   STATUS[908].EXT.ModeBit1 := FALSE;
   STATUS[908].EXT.ModeBit2 := FALSE;
   STATUS[908].EXT.ModeBit3 := FALSE;
   STATUS[908].EXT.BIT19 := FALSE;
   STATUS[908].EXT.BIT20 := FALSE;
   STATUS[908].EXT.AlarmSuppressed := FALSE;
   STATUS[908].EXT.AlarmPrsent := FALSE;
   STATUS[908].EXT.AlarmFailUnAck := FALSE;
   STATUS[908].Status := 0;
   STATUS[908].TimeStamp := 16#0000;
   STATUS[909].VALUE := 0.0;
   STATUS[909].TRIGVALUE := 0.0;
   STATUS[909].EXT.AlarmWarnUnAck := FALSE;
   STATUS[909].EXT.AckRequired := FALSE;
   STATUS[909].EXT.Maintanence := FALSE;
   STATUS[909].EXT.Operation := FALSE;
   STATUS[909].EXT.Forced := FALSE;
   STATUS[909].EXT.BIT29 := FALSE;
   STATUS[909].EXT.BIT30 := FALSE;
   STATUS[909].EXT.BIT31 := FALSE;
   STATUS[909].EXT.ModeBit1 := FALSE;
   STATUS[909].EXT.ModeBit2 := FALSE;
   STATUS[909].EXT.ModeBit3 := FALSE;
   STATUS[909].EXT.BIT19 := FALSE;
   STATUS[909].EXT.BIT20 := FALSE;
   STATUS[909].EXT.AlarmSuppressed := FALSE;
   STATUS[909].EXT.AlarmPrsent := FALSE;
   STATUS[909].EXT.AlarmFailUnAck := FALSE;
   STATUS[909].Status := 0;
   STATUS[909].TimeStamp := 16#0000;
   STATUS[910].VALUE := 0.0;
   STATUS[910].TRIGVALUE := 0.0;
   STATUS[910].EXT.AlarmWarnUnAck := FALSE;
   STATUS[910].EXT.AckRequired := FALSE;
   STATUS[910].EXT.Maintanence := FALSE;
   STATUS[910].EXT.Operation := FALSE;
   STATUS[910].EXT.Forced := FALSE;
   STATUS[910].EXT.BIT29 := FALSE;
   STATUS[910].EXT.BIT30 := FALSE;
   STATUS[910].EXT.BIT31 := FALSE;
   STATUS[910].EXT.ModeBit1 := FALSE;
   STATUS[910].EXT.ModeBit2 := FALSE;
   STATUS[910].EXT.ModeBit3 := FALSE;
   STATUS[910].EXT.BIT19 := FALSE;
   STATUS[910].EXT.BIT20 := FALSE;
   STATUS[910].EXT.AlarmSuppressed := FALSE;
   STATUS[910].EXT.AlarmPrsent := FALSE;
   STATUS[910].EXT.AlarmFailUnAck := FALSE;
   STATUS[910].Status := 0;
   STATUS[910].TimeStamp := 16#0000;
   STATUS[911].VALUE := 0.0;
   STATUS[911].TRIGVALUE := 0.0;
   STATUS[911].EXT.AlarmWarnUnAck := FALSE;
   STATUS[911].EXT.AckRequired := FALSE;
   STATUS[911].EXT.Maintanence := FALSE;
   STATUS[911].EXT.Operation := FALSE;
   STATUS[911].EXT.Forced := FALSE;
   STATUS[911].EXT.BIT29 := FALSE;
   STATUS[911].EXT.BIT30 := FALSE;
   STATUS[911].EXT.BIT31 := FALSE;
   STATUS[911].EXT.ModeBit1 := FALSE;
   STATUS[911].EXT.ModeBit2 := FALSE;
   STATUS[911].EXT.ModeBit3 := FALSE;
   STATUS[911].EXT.BIT19 := FALSE;
   STATUS[911].EXT.BIT20 := FALSE;
   STATUS[911].EXT.AlarmSuppressed := FALSE;
   STATUS[911].EXT.AlarmPrsent := FALSE;
   STATUS[911].EXT.AlarmFailUnAck := FALSE;
   STATUS[911].Status := 0;
   STATUS[911].TimeStamp := 16#0000;
   STATUS[912].VALUE := 0.0;
   STATUS[912].TRIGVALUE := 0.0;
   STATUS[912].EXT.AlarmWarnUnAck := FALSE;
   STATUS[912].EXT.AckRequired := FALSE;
   STATUS[912].EXT.Maintanence := FALSE;
   STATUS[912].EXT.Operation := FALSE;
   STATUS[912].EXT.Forced := FALSE;
   STATUS[912].EXT.BIT29 := FALSE;
   STATUS[912].EXT.BIT30 := FALSE;
   STATUS[912].EXT.BIT31 := FALSE;
   STATUS[912].EXT.ModeBit1 := FALSE;
   STATUS[912].EXT.ModeBit2 := FALSE;
   STATUS[912].EXT.ModeBit3 := FALSE;
   STATUS[912].EXT.BIT19 := FALSE;
   STATUS[912].EXT.BIT20 := FALSE;
   STATUS[912].EXT.AlarmSuppressed := FALSE;
   STATUS[912].EXT.AlarmPrsent := FALSE;
   STATUS[912].EXT.AlarmFailUnAck := FALSE;
   STATUS[912].Status := 0;
   STATUS[912].TimeStamp := 16#0000;
   STATUS[913].VALUE := 0.0;
   STATUS[913].TRIGVALUE := 0.0;
   STATUS[913].EXT.AlarmWarnUnAck := FALSE;
   STATUS[913].EXT.AckRequired := FALSE;
   STATUS[913].EXT.Maintanence := FALSE;
   STATUS[913].EXT.Operation := FALSE;
   STATUS[913].EXT.Forced := FALSE;
   STATUS[913].EXT.BIT29 := FALSE;
   STATUS[913].EXT.BIT30 := FALSE;
   STATUS[913].EXT.BIT31 := FALSE;
   STATUS[913].EXT.ModeBit1 := FALSE;
   STATUS[913].EXT.ModeBit2 := FALSE;
   STATUS[913].EXT.ModeBit3 := FALSE;
   STATUS[913].EXT.BIT19 := FALSE;
   STATUS[913].EXT.BIT20 := FALSE;
   STATUS[913].EXT.AlarmSuppressed := FALSE;
   STATUS[913].EXT.AlarmPrsent := FALSE;
   STATUS[913].EXT.AlarmFailUnAck := FALSE;
   STATUS[913].Status := 0;
   STATUS[913].TimeStamp := 16#0000;
   STATUS[914].VALUE := 0.0;
   STATUS[914].TRIGVALUE := 0.0;
   STATUS[914].EXT.AlarmWarnUnAck := FALSE;
   STATUS[914].EXT.AckRequired := FALSE;
   STATUS[914].EXT.Maintanence := FALSE;
   STATUS[914].EXT.Operation := FALSE;
   STATUS[914].EXT.Forced := FALSE;
   STATUS[914].EXT.BIT29 := FALSE;
   STATUS[914].EXT.BIT30 := FALSE;
   STATUS[914].EXT.BIT31 := FALSE;
   STATUS[914].EXT.ModeBit1 := FALSE;
   STATUS[914].EXT.ModeBit2 := FALSE;
   STATUS[914].EXT.ModeBit3 := FALSE;
   STATUS[914].EXT.BIT19 := FALSE;
   STATUS[914].EXT.BIT20 := FALSE;
   STATUS[914].EXT.AlarmSuppressed := FALSE;
   STATUS[914].EXT.AlarmPrsent := FALSE;
   STATUS[914].EXT.AlarmFailUnAck := FALSE;
   STATUS[914].Status := 0;
   STATUS[914].TimeStamp := 16#0000;
   STATUS[915].VALUE := 0.0;
   STATUS[915].TRIGVALUE := 0.0;
   STATUS[915].EXT.AlarmWarnUnAck := FALSE;
   STATUS[915].EXT.AckRequired := FALSE;
   STATUS[915].EXT.Maintanence := FALSE;
   STATUS[915].EXT.Operation := FALSE;
   STATUS[915].EXT.Forced := FALSE;
   STATUS[915].EXT.BIT29 := FALSE;
   STATUS[915].EXT.BIT30 := FALSE;
   STATUS[915].EXT.BIT31 := FALSE;
   STATUS[915].EXT.ModeBit1 := FALSE;
   STATUS[915].EXT.ModeBit2 := FALSE;
   STATUS[915].EXT.ModeBit3 := FALSE;
   STATUS[915].EXT.BIT19 := FALSE;
   STATUS[915].EXT.BIT20 := FALSE;
   STATUS[915].EXT.AlarmSuppressed := FALSE;
   STATUS[915].EXT.AlarmPrsent := FALSE;
   STATUS[915].EXT.AlarmFailUnAck := FALSE;
   STATUS[915].Status := 0;
   STATUS[915].TimeStamp := 16#0000;
   STATUS[916].VALUE := 0.0;
   STATUS[916].TRIGVALUE := 0.0;
   STATUS[916].EXT.AlarmWarnUnAck := FALSE;
   STATUS[916].EXT.AckRequired := FALSE;
   STATUS[916].EXT.Maintanence := FALSE;
   STATUS[916].EXT.Operation := FALSE;
   STATUS[916].EXT.Forced := FALSE;
   STATUS[916].EXT.BIT29 := FALSE;
   STATUS[916].EXT.BIT30 := FALSE;
   STATUS[916].EXT.BIT31 := FALSE;
   STATUS[916].EXT.ModeBit1 := FALSE;
   STATUS[916].EXT.ModeBit2 := FALSE;
   STATUS[916].EXT.ModeBit3 := FALSE;
   STATUS[916].EXT.BIT19 := FALSE;
   STATUS[916].EXT.BIT20 := FALSE;
   STATUS[916].EXT.AlarmSuppressed := FALSE;
   STATUS[916].EXT.AlarmPrsent := FALSE;
   STATUS[916].EXT.AlarmFailUnAck := FALSE;
   STATUS[916].Status := 0;
   STATUS[916].TimeStamp := 16#0000;
   STATUS[917].VALUE := 0.0;
   STATUS[917].TRIGVALUE := 0.0;
   STATUS[917].EXT.AlarmWarnUnAck := FALSE;
   STATUS[917].EXT.AckRequired := FALSE;
   STATUS[917].EXT.Maintanence := FALSE;
   STATUS[917].EXT.Operation := FALSE;
   STATUS[917].EXT.Forced := FALSE;
   STATUS[917].EXT.BIT29 := FALSE;
   STATUS[917].EXT.BIT30 := FALSE;
   STATUS[917].EXT.BIT31 := FALSE;
   STATUS[917].EXT.ModeBit1 := FALSE;
   STATUS[917].EXT.ModeBit2 := FALSE;
   STATUS[917].EXT.ModeBit3 := FALSE;
   STATUS[917].EXT.BIT19 := FALSE;
   STATUS[917].EXT.BIT20 := FALSE;
   STATUS[917].EXT.AlarmSuppressed := FALSE;
   STATUS[917].EXT.AlarmPrsent := FALSE;
   STATUS[917].EXT.AlarmFailUnAck := FALSE;
   STATUS[917].Status := 0;
   STATUS[917].TimeStamp := 16#0000;
   STATUS[918].VALUE := 0.0;
   STATUS[918].TRIGVALUE := 0.0;
   STATUS[918].EXT.AlarmWarnUnAck := FALSE;
   STATUS[918].EXT.AckRequired := FALSE;
   STATUS[918].EXT.Maintanence := FALSE;
   STATUS[918].EXT.Operation := FALSE;
   STATUS[918].EXT.Forced := FALSE;
   STATUS[918].EXT.BIT29 := FALSE;
   STATUS[918].EXT.BIT30 := FALSE;
   STATUS[918].EXT.BIT31 := FALSE;
   STATUS[918].EXT.ModeBit1 := FALSE;
   STATUS[918].EXT.ModeBit2 := FALSE;
   STATUS[918].EXT.ModeBit3 := FALSE;
   STATUS[918].EXT.BIT19 := FALSE;
   STATUS[918].EXT.BIT20 := FALSE;
   STATUS[918].EXT.AlarmSuppressed := FALSE;
   STATUS[918].EXT.AlarmPrsent := FALSE;
   STATUS[918].EXT.AlarmFailUnAck := FALSE;
   STATUS[918].Status := 0;
   STATUS[918].TimeStamp := 16#0000;
   STATUS[919].VALUE := 0.0;
   STATUS[919].TRIGVALUE := 0.0;
   STATUS[919].EXT.AlarmWarnUnAck := FALSE;
   STATUS[919].EXT.AckRequired := FALSE;
   STATUS[919].EXT.Maintanence := FALSE;
   STATUS[919].EXT.Operation := FALSE;
   STATUS[919].EXT.Forced := FALSE;
   STATUS[919].EXT.BIT29 := FALSE;
   STATUS[919].EXT.BIT30 := FALSE;
   STATUS[919].EXT.BIT31 := FALSE;
   STATUS[919].EXT.ModeBit1 := FALSE;
   STATUS[919].EXT.ModeBit2 := FALSE;
   STATUS[919].EXT.ModeBit3 := FALSE;
   STATUS[919].EXT.BIT19 := FALSE;
   STATUS[919].EXT.BIT20 := FALSE;
   STATUS[919].EXT.AlarmSuppressed := FALSE;
   STATUS[919].EXT.AlarmPrsent := FALSE;
   STATUS[919].EXT.AlarmFailUnAck := FALSE;
   STATUS[919].Status := 0;
   STATUS[919].TimeStamp := 16#0000;
   STATUS[920].VALUE := 0.0;
   STATUS[920].TRIGVALUE := 0.0;
   STATUS[920].EXT.AlarmWarnUnAck := FALSE;
   STATUS[920].EXT.AckRequired := FALSE;
   STATUS[920].EXT.Maintanence := FALSE;
   STATUS[920].EXT.Operation := FALSE;
   STATUS[920].EXT.Forced := FALSE;
   STATUS[920].EXT.BIT29 := FALSE;
   STATUS[920].EXT.BIT30 := FALSE;
   STATUS[920].EXT.BIT31 := FALSE;
   STATUS[920].EXT.ModeBit1 := FALSE;
   STATUS[920].EXT.ModeBit2 := FALSE;
   STATUS[920].EXT.ModeBit3 := FALSE;
   STATUS[920].EXT.BIT19 := FALSE;
   STATUS[920].EXT.BIT20 := FALSE;
   STATUS[920].EXT.AlarmSuppressed := FALSE;
   STATUS[920].EXT.AlarmPrsent := FALSE;
   STATUS[920].EXT.AlarmFailUnAck := FALSE;
   STATUS[920].Status := 0;
   STATUS[920].TimeStamp := 16#0000;
   STATUS[921].VALUE := 0.0;
   STATUS[921].TRIGVALUE := 0.0;
   STATUS[921].EXT.AlarmWarnUnAck := FALSE;
   STATUS[921].EXT.AckRequired := FALSE;
   STATUS[921].EXT.Maintanence := FALSE;
   STATUS[921].EXT.Operation := FALSE;
   STATUS[921].EXT.Forced := FALSE;
   STATUS[921].EXT.BIT29 := FALSE;
   STATUS[921].EXT.BIT30 := FALSE;
   STATUS[921].EXT.BIT31 := FALSE;
   STATUS[921].EXT.ModeBit1 := FALSE;
   STATUS[921].EXT.ModeBit2 := FALSE;
   STATUS[921].EXT.ModeBit3 := FALSE;
   STATUS[921].EXT.BIT19 := FALSE;
   STATUS[921].EXT.BIT20 := FALSE;
   STATUS[921].EXT.AlarmSuppressed := FALSE;
   STATUS[921].EXT.AlarmPrsent := FALSE;
   STATUS[921].EXT.AlarmFailUnAck := FALSE;
   STATUS[921].Status := 0;
   STATUS[921].TimeStamp := 16#0000;
   STATUS[922].VALUE := 0.0;
   STATUS[922].TRIGVALUE := 0.0;
   STATUS[922].EXT.AlarmWarnUnAck := FALSE;
   STATUS[922].EXT.AckRequired := FALSE;
   STATUS[922].EXT.Maintanence := FALSE;
   STATUS[922].EXT.Operation := FALSE;
   STATUS[922].EXT.Forced := FALSE;
   STATUS[922].EXT.BIT29 := FALSE;
   STATUS[922].EXT.BIT30 := FALSE;
   STATUS[922].EXT.BIT31 := FALSE;
   STATUS[922].EXT.ModeBit1 := FALSE;
   STATUS[922].EXT.ModeBit2 := FALSE;
   STATUS[922].EXT.ModeBit3 := FALSE;
   STATUS[922].EXT.BIT19 := FALSE;
   STATUS[922].EXT.BIT20 := FALSE;
   STATUS[922].EXT.AlarmSuppressed := FALSE;
   STATUS[922].EXT.AlarmPrsent := FALSE;
   STATUS[922].EXT.AlarmFailUnAck := FALSE;
   STATUS[922].Status := 0;
   STATUS[922].TimeStamp := 16#0000;
   STATUS[923].VALUE := 0.0;
   STATUS[923].TRIGVALUE := 0.0;
   STATUS[923].EXT.AlarmWarnUnAck := FALSE;
   STATUS[923].EXT.AckRequired := FALSE;
   STATUS[923].EXT.Maintanence := FALSE;
   STATUS[923].EXT.Operation := FALSE;
   STATUS[923].EXT.Forced := FALSE;
   STATUS[923].EXT.BIT29 := FALSE;
   STATUS[923].EXT.BIT30 := FALSE;
   STATUS[923].EXT.BIT31 := FALSE;
   STATUS[923].EXT.ModeBit1 := FALSE;
   STATUS[923].EXT.ModeBit2 := FALSE;
   STATUS[923].EXT.ModeBit3 := FALSE;
   STATUS[923].EXT.BIT19 := FALSE;
   STATUS[923].EXT.BIT20 := FALSE;
   STATUS[923].EXT.AlarmSuppressed := FALSE;
   STATUS[923].EXT.AlarmPrsent := FALSE;
   STATUS[923].EXT.AlarmFailUnAck := FALSE;
   STATUS[923].Status := 0;
   STATUS[923].TimeStamp := 16#0000;
   STATUS[924].VALUE := 0.0;
   STATUS[924].TRIGVALUE := 0.0;
   STATUS[924].EXT.AlarmWarnUnAck := FALSE;
   STATUS[924].EXT.AckRequired := FALSE;
   STATUS[924].EXT.Maintanence := FALSE;
   STATUS[924].EXT.Operation := FALSE;
   STATUS[924].EXT.Forced := FALSE;
   STATUS[924].EXT.BIT29 := FALSE;
   STATUS[924].EXT.BIT30 := FALSE;
   STATUS[924].EXT.BIT31 := FALSE;
   STATUS[924].EXT.ModeBit1 := FALSE;
   STATUS[924].EXT.ModeBit2 := FALSE;
   STATUS[924].EXT.ModeBit3 := FALSE;
   STATUS[924].EXT.BIT19 := FALSE;
   STATUS[924].EXT.BIT20 := FALSE;
   STATUS[924].EXT.AlarmSuppressed := FALSE;
   STATUS[924].EXT.AlarmPrsent := FALSE;
   STATUS[924].EXT.AlarmFailUnAck := FALSE;
   STATUS[924].Status := 0;
   STATUS[924].TimeStamp := 16#0000;
   STATUS[925].VALUE := 0.0;
   STATUS[925].TRIGVALUE := 0.0;
   STATUS[925].EXT.AlarmWarnUnAck := FALSE;
   STATUS[925].EXT.AckRequired := FALSE;
   STATUS[925].EXT.Maintanence := FALSE;
   STATUS[925].EXT.Operation := FALSE;
   STATUS[925].EXT.Forced := FALSE;
   STATUS[925].EXT.BIT29 := FALSE;
   STATUS[925].EXT.BIT30 := FALSE;
   STATUS[925].EXT.BIT31 := FALSE;
   STATUS[925].EXT.ModeBit1 := FALSE;
   STATUS[925].EXT.ModeBit2 := FALSE;
   STATUS[925].EXT.ModeBit3 := FALSE;
   STATUS[925].EXT.BIT19 := FALSE;
   STATUS[925].EXT.BIT20 := FALSE;
   STATUS[925].EXT.AlarmSuppressed := FALSE;
   STATUS[925].EXT.AlarmPrsent := FALSE;
   STATUS[925].EXT.AlarmFailUnAck := FALSE;
   STATUS[925].Status := 0;
   STATUS[925].TimeStamp := 16#0000;
   STATUS[926].VALUE := 0.0;
   STATUS[926].TRIGVALUE := 0.0;
   STATUS[926].EXT.AlarmWarnUnAck := FALSE;
   STATUS[926].EXT.AckRequired := FALSE;
   STATUS[926].EXT.Maintanence := FALSE;
   STATUS[926].EXT.Operation := FALSE;
   STATUS[926].EXT.Forced := FALSE;
   STATUS[926].EXT.BIT29 := FALSE;
   STATUS[926].EXT.BIT30 := FALSE;
   STATUS[926].EXT.BIT31 := FALSE;
   STATUS[926].EXT.ModeBit1 := FALSE;
   STATUS[926].EXT.ModeBit2 := FALSE;
   STATUS[926].EXT.ModeBit3 := FALSE;
   STATUS[926].EXT.BIT19 := FALSE;
   STATUS[926].EXT.BIT20 := FALSE;
   STATUS[926].EXT.AlarmSuppressed := FALSE;
   STATUS[926].EXT.AlarmPrsent := FALSE;
   STATUS[926].EXT.AlarmFailUnAck := FALSE;
   STATUS[926].Status := 0;
   STATUS[926].TimeStamp := 16#0000;
   STATUS[927].VALUE := 0.0;
   STATUS[927].TRIGVALUE := 0.0;
   STATUS[927].EXT.AlarmWarnUnAck := FALSE;
   STATUS[927].EXT.AckRequired := FALSE;
   STATUS[927].EXT.Maintanence := FALSE;
   STATUS[927].EXT.Operation := FALSE;
   STATUS[927].EXT.Forced := FALSE;
   STATUS[927].EXT.BIT29 := FALSE;
   STATUS[927].EXT.BIT30 := FALSE;
   STATUS[927].EXT.BIT31 := FALSE;
   STATUS[927].EXT.ModeBit1 := FALSE;
   STATUS[927].EXT.ModeBit2 := FALSE;
   STATUS[927].EXT.ModeBit3 := FALSE;
   STATUS[927].EXT.BIT19 := FALSE;
   STATUS[927].EXT.BIT20 := FALSE;
   STATUS[927].EXT.AlarmSuppressed := FALSE;
   STATUS[927].EXT.AlarmPrsent := FALSE;
   STATUS[927].EXT.AlarmFailUnAck := FALSE;
   STATUS[927].Status := 0;
   STATUS[927].TimeStamp := 16#0000;
   STATUS[928].VALUE := 0.0;
   STATUS[928].TRIGVALUE := 0.0;
   STATUS[928].EXT.AlarmWarnUnAck := FALSE;
   STATUS[928].EXT.AckRequired := FALSE;
   STATUS[928].EXT.Maintanence := FALSE;
   STATUS[928].EXT.Operation := FALSE;
   STATUS[928].EXT.Forced := FALSE;
   STATUS[928].EXT.BIT29 := FALSE;
   STATUS[928].EXT.BIT30 := FALSE;
   STATUS[928].EXT.BIT31 := FALSE;
   STATUS[928].EXT.ModeBit1 := FALSE;
   STATUS[928].EXT.ModeBit2 := FALSE;
   STATUS[928].EXT.ModeBit3 := FALSE;
   STATUS[928].EXT.BIT19 := FALSE;
   STATUS[928].EXT.BIT20 := FALSE;
   STATUS[928].EXT.AlarmSuppressed := FALSE;
   STATUS[928].EXT.AlarmPrsent := FALSE;
   STATUS[928].EXT.AlarmFailUnAck := FALSE;
   STATUS[928].Status := 0;
   STATUS[928].TimeStamp := 16#0000;
   STATUS[929].VALUE := 0.0;
   STATUS[929].TRIGVALUE := 0.0;
   STATUS[929].EXT.AlarmWarnUnAck := FALSE;
   STATUS[929].EXT.AckRequired := FALSE;
   STATUS[929].EXT.Maintanence := FALSE;
   STATUS[929].EXT.Operation := FALSE;
   STATUS[929].EXT.Forced := FALSE;
   STATUS[929].EXT.BIT29 := FALSE;
   STATUS[929].EXT.BIT30 := FALSE;
   STATUS[929].EXT.BIT31 := FALSE;
   STATUS[929].EXT.ModeBit1 := FALSE;
   STATUS[929].EXT.ModeBit2 := FALSE;
   STATUS[929].EXT.ModeBit3 := FALSE;
   STATUS[929].EXT.BIT19 := FALSE;
   STATUS[929].EXT.BIT20 := FALSE;
   STATUS[929].EXT.AlarmSuppressed := FALSE;
   STATUS[929].EXT.AlarmPrsent := FALSE;
   STATUS[929].EXT.AlarmFailUnAck := FALSE;
   STATUS[929].Status := 0;
   STATUS[929].TimeStamp := 16#0000;
   STATUS[930].VALUE := 0.0;
   STATUS[930].TRIGVALUE := 0.0;
   STATUS[930].EXT.AlarmWarnUnAck := FALSE;
   STATUS[930].EXT.AckRequired := FALSE;
   STATUS[930].EXT.Maintanence := FALSE;
   STATUS[930].EXT.Operation := FALSE;
   STATUS[930].EXT.Forced := FALSE;
   STATUS[930].EXT.BIT29 := FALSE;
   STATUS[930].EXT.BIT30 := FALSE;
   STATUS[930].EXT.BIT31 := FALSE;
   STATUS[930].EXT.ModeBit1 := FALSE;
   STATUS[930].EXT.ModeBit2 := FALSE;
   STATUS[930].EXT.ModeBit3 := FALSE;
   STATUS[930].EXT.BIT19 := FALSE;
   STATUS[930].EXT.BIT20 := FALSE;
   STATUS[930].EXT.AlarmSuppressed := FALSE;
   STATUS[930].EXT.AlarmPrsent := FALSE;
   STATUS[930].EXT.AlarmFailUnAck := FALSE;
   STATUS[930].Status := 0;
   STATUS[930].TimeStamp := 16#0000;
   STATUS[931].VALUE := 0.0;
   STATUS[931].TRIGVALUE := 0.0;
   STATUS[931].EXT.AlarmWarnUnAck := FALSE;
   STATUS[931].EXT.AckRequired := FALSE;
   STATUS[931].EXT.Maintanence := FALSE;
   STATUS[931].EXT.Operation := FALSE;
   STATUS[931].EXT.Forced := FALSE;
   STATUS[931].EXT.BIT29 := FALSE;
   STATUS[931].EXT.BIT30 := FALSE;
   STATUS[931].EXT.BIT31 := FALSE;
   STATUS[931].EXT.ModeBit1 := FALSE;
   STATUS[931].EXT.ModeBit2 := FALSE;
   STATUS[931].EXT.ModeBit3 := FALSE;
   STATUS[931].EXT.BIT19 := FALSE;
   STATUS[931].EXT.BIT20 := FALSE;
   STATUS[931].EXT.AlarmSuppressed := FALSE;
   STATUS[931].EXT.AlarmPrsent := FALSE;
   STATUS[931].EXT.AlarmFailUnAck := FALSE;
   STATUS[931].Status := 0;
   STATUS[931].TimeStamp := 16#0000;
   STATUS[932].VALUE := 0.0;
   STATUS[932].TRIGVALUE := 0.0;
   STATUS[932].EXT.AlarmWarnUnAck := FALSE;
   STATUS[932].EXT.AckRequired := FALSE;
   STATUS[932].EXT.Maintanence := FALSE;
   STATUS[932].EXT.Operation := FALSE;
   STATUS[932].EXT.Forced := FALSE;
   STATUS[932].EXT.BIT29 := FALSE;
   STATUS[932].EXT.BIT30 := FALSE;
   STATUS[932].EXT.BIT31 := FALSE;
   STATUS[932].EXT.ModeBit1 := FALSE;
   STATUS[932].EXT.ModeBit2 := FALSE;
   STATUS[932].EXT.ModeBit3 := FALSE;
   STATUS[932].EXT.BIT19 := FALSE;
   STATUS[932].EXT.BIT20 := FALSE;
   STATUS[932].EXT.AlarmSuppressed := FALSE;
   STATUS[932].EXT.AlarmPrsent := FALSE;
   STATUS[932].EXT.AlarmFailUnAck := FALSE;
   STATUS[932].Status := 0;
   STATUS[932].TimeStamp := 16#0000;
   STATUS[933].VALUE := 0.0;
   STATUS[933].TRIGVALUE := 0.0;
   STATUS[933].EXT.AlarmWarnUnAck := FALSE;
   STATUS[933].EXT.AckRequired := FALSE;
   STATUS[933].EXT.Maintanence := FALSE;
   STATUS[933].EXT.Operation := FALSE;
   STATUS[933].EXT.Forced := FALSE;
   STATUS[933].EXT.BIT29 := FALSE;
   STATUS[933].EXT.BIT30 := FALSE;
   STATUS[933].EXT.BIT31 := FALSE;
   STATUS[933].EXT.ModeBit1 := FALSE;
   STATUS[933].EXT.ModeBit2 := FALSE;
   STATUS[933].EXT.ModeBit3 := FALSE;
   STATUS[933].EXT.BIT19 := FALSE;
   STATUS[933].EXT.BIT20 := FALSE;
   STATUS[933].EXT.AlarmSuppressed := FALSE;
   STATUS[933].EXT.AlarmPrsent := FALSE;
   STATUS[933].EXT.AlarmFailUnAck := FALSE;
   STATUS[933].Status := 0;
   STATUS[933].TimeStamp := 16#0000;
   STATUS[934].VALUE := 0.0;
   STATUS[934].TRIGVALUE := 0.0;
   STATUS[934].EXT.AlarmWarnUnAck := FALSE;
   STATUS[934].EXT.AckRequired := FALSE;
   STATUS[934].EXT.Maintanence := FALSE;
   STATUS[934].EXT.Operation := FALSE;
   STATUS[934].EXT.Forced := FALSE;
   STATUS[934].EXT.BIT29 := FALSE;
   STATUS[934].EXT.BIT30 := FALSE;
   STATUS[934].EXT.BIT31 := FALSE;
   STATUS[934].EXT.ModeBit1 := FALSE;
   STATUS[934].EXT.ModeBit2 := FALSE;
   STATUS[934].EXT.ModeBit3 := FALSE;
   STATUS[934].EXT.BIT19 := FALSE;
   STATUS[934].EXT.BIT20 := FALSE;
   STATUS[934].EXT.AlarmSuppressed := FALSE;
   STATUS[934].EXT.AlarmPrsent := FALSE;
   STATUS[934].EXT.AlarmFailUnAck := FALSE;
   STATUS[934].Status := 0;
   STATUS[934].TimeStamp := 16#0000;
   STATUS[935].VALUE := 0.0;
   STATUS[935].TRIGVALUE := 0.0;
   STATUS[935].EXT.AlarmWarnUnAck := FALSE;
   STATUS[935].EXT.AckRequired := FALSE;
   STATUS[935].EXT.Maintanence := FALSE;
   STATUS[935].EXT.Operation := FALSE;
   STATUS[935].EXT.Forced := FALSE;
   STATUS[935].EXT.BIT29 := FALSE;
   STATUS[935].EXT.BIT30 := FALSE;
   STATUS[935].EXT.BIT31 := FALSE;
   STATUS[935].EXT.ModeBit1 := FALSE;
   STATUS[935].EXT.ModeBit2 := FALSE;
   STATUS[935].EXT.ModeBit3 := FALSE;
   STATUS[935].EXT.BIT19 := FALSE;
   STATUS[935].EXT.BIT20 := FALSE;
   STATUS[935].EXT.AlarmSuppressed := FALSE;
   STATUS[935].EXT.AlarmPrsent := FALSE;
   STATUS[935].EXT.AlarmFailUnAck := FALSE;
   STATUS[935].Status := 0;
   STATUS[935].TimeStamp := 16#0000;
   STATUS[936].VALUE := 0.0;
   STATUS[936].TRIGVALUE := 0.0;
   STATUS[936].EXT.AlarmWarnUnAck := FALSE;
   STATUS[936].EXT.AckRequired := FALSE;
   STATUS[936].EXT.Maintanence := FALSE;
   STATUS[936].EXT.Operation := FALSE;
   STATUS[936].EXT.Forced := FALSE;
   STATUS[936].EXT.BIT29 := FALSE;
   STATUS[936].EXT.BIT30 := FALSE;
   STATUS[936].EXT.BIT31 := FALSE;
   STATUS[936].EXT.ModeBit1 := FALSE;
   STATUS[936].EXT.ModeBit2 := FALSE;
   STATUS[936].EXT.ModeBit3 := FALSE;
   STATUS[936].EXT.BIT19 := FALSE;
   STATUS[936].EXT.BIT20 := FALSE;
   STATUS[936].EXT.AlarmSuppressed := FALSE;
   STATUS[936].EXT.AlarmPrsent := FALSE;
   STATUS[936].EXT.AlarmFailUnAck := FALSE;
   STATUS[936].Status := 0;
   STATUS[936].TimeStamp := 16#0000;
   STATUS[937].VALUE := 0.0;
   STATUS[937].TRIGVALUE := 0.0;
   STATUS[937].EXT.AlarmWarnUnAck := FALSE;
   STATUS[937].EXT.AckRequired := FALSE;
   STATUS[937].EXT.Maintanence := FALSE;
   STATUS[937].EXT.Operation := FALSE;
   STATUS[937].EXT.Forced := FALSE;
   STATUS[937].EXT.BIT29 := FALSE;
   STATUS[937].EXT.BIT30 := FALSE;
   STATUS[937].EXT.BIT31 := FALSE;
   STATUS[937].EXT.ModeBit1 := FALSE;
   STATUS[937].EXT.ModeBit2 := FALSE;
   STATUS[937].EXT.ModeBit3 := FALSE;
   STATUS[937].EXT.BIT19 := FALSE;
   STATUS[937].EXT.BIT20 := FALSE;
   STATUS[937].EXT.AlarmSuppressed := FALSE;
   STATUS[937].EXT.AlarmPrsent := FALSE;
   STATUS[937].EXT.AlarmFailUnAck := FALSE;
   STATUS[937].Status := 0;
   STATUS[937].TimeStamp := 16#0000;
   STATUS[938].VALUE := 0.0;
   STATUS[938].TRIGVALUE := 0.0;
   STATUS[938].EXT.AlarmWarnUnAck := FALSE;
   STATUS[938].EXT.AckRequired := FALSE;
   STATUS[938].EXT.Maintanence := FALSE;
   STATUS[938].EXT.Operation := FALSE;
   STATUS[938].EXT.Forced := FALSE;
   STATUS[938].EXT.BIT29 := FALSE;
   STATUS[938].EXT.BIT30 := FALSE;
   STATUS[938].EXT.BIT31 := FALSE;
   STATUS[938].EXT.ModeBit1 := FALSE;
   STATUS[938].EXT.ModeBit2 := FALSE;
   STATUS[938].EXT.ModeBit3 := FALSE;
   STATUS[938].EXT.BIT19 := FALSE;
   STATUS[938].EXT.BIT20 := FALSE;
   STATUS[938].EXT.AlarmSuppressed := FALSE;
   STATUS[938].EXT.AlarmPrsent := FALSE;
   STATUS[938].EXT.AlarmFailUnAck := FALSE;
   STATUS[938].Status := 0;
   STATUS[938].TimeStamp := 16#0000;
   STATUS[939].VALUE := 0.0;
   STATUS[939].TRIGVALUE := 0.0;
   STATUS[939].EXT.AlarmWarnUnAck := FALSE;
   STATUS[939].EXT.AckRequired := FALSE;
   STATUS[939].EXT.Maintanence := FALSE;
   STATUS[939].EXT.Operation := FALSE;
   STATUS[939].EXT.Forced := FALSE;
   STATUS[939].EXT.BIT29 := FALSE;
   STATUS[939].EXT.BIT30 := FALSE;
   STATUS[939].EXT.BIT31 := FALSE;
   STATUS[939].EXT.ModeBit1 := FALSE;
   STATUS[939].EXT.ModeBit2 := FALSE;
   STATUS[939].EXT.ModeBit3 := FALSE;
   STATUS[939].EXT.BIT19 := FALSE;
   STATUS[939].EXT.BIT20 := FALSE;
   STATUS[939].EXT.AlarmSuppressed := FALSE;
   STATUS[939].EXT.AlarmPrsent := FALSE;
   STATUS[939].EXT.AlarmFailUnAck := FALSE;
   STATUS[939].Status := 0;
   STATUS[939].TimeStamp := 16#0000;
   STATUS[940].VALUE := 0.0;
   STATUS[940].TRIGVALUE := 0.0;
   STATUS[940].EXT.AlarmWarnUnAck := FALSE;
   STATUS[940].EXT.AckRequired := FALSE;
   STATUS[940].EXT.Maintanence := FALSE;
   STATUS[940].EXT.Operation := FALSE;
   STATUS[940].EXT.Forced := FALSE;
   STATUS[940].EXT.BIT29 := FALSE;
   STATUS[940].EXT.BIT30 := FALSE;
   STATUS[940].EXT.BIT31 := FALSE;
   STATUS[940].EXT.ModeBit1 := FALSE;
   STATUS[940].EXT.ModeBit2 := FALSE;
   STATUS[940].EXT.ModeBit3 := FALSE;
   STATUS[940].EXT.BIT19 := FALSE;
   STATUS[940].EXT.BIT20 := FALSE;
   STATUS[940].EXT.AlarmSuppressed := FALSE;
   STATUS[940].EXT.AlarmPrsent := FALSE;
   STATUS[940].EXT.AlarmFailUnAck := FALSE;
   STATUS[940].Status := 0;
   STATUS[940].TimeStamp := 16#0000;
   STATUS[941].VALUE := 0.0;
   STATUS[941].TRIGVALUE := 0.0;
   STATUS[941].EXT.AlarmWarnUnAck := FALSE;
   STATUS[941].EXT.AckRequired := FALSE;
   STATUS[941].EXT.Maintanence := FALSE;
   STATUS[941].EXT.Operation := FALSE;
   STATUS[941].EXT.Forced := FALSE;
   STATUS[941].EXT.BIT29 := FALSE;
   STATUS[941].EXT.BIT30 := FALSE;
   STATUS[941].EXT.BIT31 := FALSE;
   STATUS[941].EXT.ModeBit1 := FALSE;
   STATUS[941].EXT.ModeBit2 := FALSE;
   STATUS[941].EXT.ModeBit3 := FALSE;
   STATUS[941].EXT.BIT19 := FALSE;
   STATUS[941].EXT.BIT20 := FALSE;
   STATUS[941].EXT.AlarmSuppressed := FALSE;
   STATUS[941].EXT.AlarmPrsent := FALSE;
   STATUS[941].EXT.AlarmFailUnAck := FALSE;
   STATUS[941].Status := 0;
   STATUS[941].TimeStamp := 16#0000;
   STATUS[942].VALUE := 0.0;
   STATUS[942].TRIGVALUE := 0.0;
   STATUS[942].EXT.AlarmWarnUnAck := FALSE;
   STATUS[942].EXT.AckRequired := FALSE;
   STATUS[942].EXT.Maintanence := FALSE;
   STATUS[942].EXT.Operation := FALSE;
   STATUS[942].EXT.Forced := FALSE;
   STATUS[942].EXT.BIT29 := FALSE;
   STATUS[942].EXT.BIT30 := FALSE;
   STATUS[942].EXT.BIT31 := FALSE;
   STATUS[942].EXT.ModeBit1 := FALSE;
   STATUS[942].EXT.ModeBit2 := FALSE;
   STATUS[942].EXT.ModeBit3 := FALSE;
   STATUS[942].EXT.BIT19 := FALSE;
   STATUS[942].EXT.BIT20 := FALSE;
   STATUS[942].EXT.AlarmSuppressed := FALSE;
   STATUS[942].EXT.AlarmPrsent := FALSE;
   STATUS[942].EXT.AlarmFailUnAck := FALSE;
   STATUS[942].Status := 0;
   STATUS[942].TimeStamp := 16#0000;
   STATUS[943].VALUE := 0.0;
   STATUS[943].TRIGVALUE := 0.0;
   STATUS[943].EXT.AlarmWarnUnAck := FALSE;
   STATUS[943].EXT.AckRequired := FALSE;
   STATUS[943].EXT.Maintanence := FALSE;
   STATUS[943].EXT.Operation := FALSE;
   STATUS[943].EXT.Forced := FALSE;
   STATUS[943].EXT.BIT29 := FALSE;
   STATUS[943].EXT.BIT30 := FALSE;
   STATUS[943].EXT.BIT31 := FALSE;
   STATUS[943].EXT.ModeBit1 := FALSE;
   STATUS[943].EXT.ModeBit2 := FALSE;
   STATUS[943].EXT.ModeBit3 := FALSE;
   STATUS[943].EXT.BIT19 := FALSE;
   STATUS[943].EXT.BIT20 := FALSE;
   STATUS[943].EXT.AlarmSuppressed := FALSE;
   STATUS[943].EXT.AlarmPrsent := FALSE;
   STATUS[943].EXT.AlarmFailUnAck := FALSE;
   STATUS[943].Status := 0;
   STATUS[943].TimeStamp := 16#0000;
   STATUS[944].VALUE := 0.0;
   STATUS[944].TRIGVALUE := 0.0;
   STATUS[944].EXT.AlarmWarnUnAck := FALSE;
   STATUS[944].EXT.AckRequired := FALSE;
   STATUS[944].EXT.Maintanence := FALSE;
   STATUS[944].EXT.Operation := FALSE;
   STATUS[944].EXT.Forced := FALSE;
   STATUS[944].EXT.BIT29 := FALSE;
   STATUS[944].EXT.BIT30 := FALSE;
   STATUS[944].EXT.BIT31 := FALSE;
   STATUS[944].EXT.ModeBit1 := FALSE;
   STATUS[944].EXT.ModeBit2 := FALSE;
   STATUS[944].EXT.ModeBit3 := FALSE;
   STATUS[944].EXT.BIT19 := FALSE;
   STATUS[944].EXT.BIT20 := FALSE;
   STATUS[944].EXT.AlarmSuppressed := FALSE;
   STATUS[944].EXT.AlarmPrsent := FALSE;
   STATUS[944].EXT.AlarmFailUnAck := FALSE;
   STATUS[944].Status := 0;
   STATUS[944].TimeStamp := 16#0000;
   STATUS[945].VALUE := 0.0;
   STATUS[945].TRIGVALUE := 0.0;
   STATUS[945].EXT.AlarmWarnUnAck := FALSE;
   STATUS[945].EXT.AckRequired := FALSE;
   STATUS[945].EXT.Maintanence := FALSE;
   STATUS[945].EXT.Operation := FALSE;
   STATUS[945].EXT.Forced := FALSE;
   STATUS[945].EXT.BIT29 := FALSE;
   STATUS[945].EXT.BIT30 := FALSE;
   STATUS[945].EXT.BIT31 := FALSE;
   STATUS[945].EXT.ModeBit1 := FALSE;
   STATUS[945].EXT.ModeBit2 := FALSE;
   STATUS[945].EXT.ModeBit3 := FALSE;
   STATUS[945].EXT.BIT19 := FALSE;
   STATUS[945].EXT.BIT20 := FALSE;
   STATUS[945].EXT.AlarmSuppressed := FALSE;
   STATUS[945].EXT.AlarmPrsent := FALSE;
   STATUS[945].EXT.AlarmFailUnAck := FALSE;
   STATUS[945].Status := 0;
   STATUS[945].TimeStamp := 16#0000;
   STATUS[946].VALUE := 0.0;
   STATUS[946].TRIGVALUE := 0.0;
   STATUS[946].EXT.AlarmWarnUnAck := FALSE;
   STATUS[946].EXT.AckRequired := FALSE;
   STATUS[946].EXT.Maintanence := FALSE;
   STATUS[946].EXT.Operation := FALSE;
   STATUS[946].EXT.Forced := FALSE;
   STATUS[946].EXT.BIT29 := FALSE;
   STATUS[946].EXT.BIT30 := FALSE;
   STATUS[946].EXT.BIT31 := FALSE;
   STATUS[946].EXT.ModeBit1 := FALSE;
   STATUS[946].EXT.ModeBit2 := FALSE;
   STATUS[946].EXT.ModeBit3 := FALSE;
   STATUS[946].EXT.BIT19 := FALSE;
   STATUS[946].EXT.BIT20 := FALSE;
   STATUS[946].EXT.AlarmSuppressed := FALSE;
   STATUS[946].EXT.AlarmPrsent := FALSE;
   STATUS[946].EXT.AlarmFailUnAck := FALSE;
   STATUS[946].Status := 0;
   STATUS[946].TimeStamp := 16#0000;
   STATUS[947].VALUE := 0.0;
   STATUS[947].TRIGVALUE := 0.0;
   STATUS[947].EXT.AlarmWarnUnAck := FALSE;
   STATUS[947].EXT.AckRequired := FALSE;
   STATUS[947].EXT.Maintanence := FALSE;
   STATUS[947].EXT.Operation := FALSE;
   STATUS[947].EXT.Forced := FALSE;
   STATUS[947].EXT.BIT29 := FALSE;
   STATUS[947].EXT.BIT30 := FALSE;
   STATUS[947].EXT.BIT31 := FALSE;
   STATUS[947].EXT.ModeBit1 := FALSE;
   STATUS[947].EXT.ModeBit2 := FALSE;
   STATUS[947].EXT.ModeBit3 := FALSE;
   STATUS[947].EXT.BIT19 := FALSE;
   STATUS[947].EXT.BIT20 := FALSE;
   STATUS[947].EXT.AlarmSuppressed := FALSE;
   STATUS[947].EXT.AlarmPrsent := FALSE;
   STATUS[947].EXT.AlarmFailUnAck := FALSE;
   STATUS[947].Status := 0;
   STATUS[947].TimeStamp := 16#0000;
   STATUS[948].VALUE := 0.0;
   STATUS[948].TRIGVALUE := 0.0;
   STATUS[948].EXT.AlarmWarnUnAck := FALSE;
   STATUS[948].EXT.AckRequired := FALSE;
   STATUS[948].EXT.Maintanence := FALSE;
   STATUS[948].EXT.Operation := FALSE;
   STATUS[948].EXT.Forced := FALSE;
   STATUS[948].EXT.BIT29 := FALSE;
   STATUS[948].EXT.BIT30 := FALSE;
   STATUS[948].EXT.BIT31 := FALSE;
   STATUS[948].EXT.ModeBit1 := FALSE;
   STATUS[948].EXT.ModeBit2 := FALSE;
   STATUS[948].EXT.ModeBit3 := FALSE;
   STATUS[948].EXT.BIT19 := FALSE;
   STATUS[948].EXT.BIT20 := FALSE;
   STATUS[948].EXT.AlarmSuppressed := FALSE;
   STATUS[948].EXT.AlarmPrsent := FALSE;
   STATUS[948].EXT.AlarmFailUnAck := FALSE;
   STATUS[948].Status := 0;
   STATUS[948].TimeStamp := 16#0000;
   STATUS[949].VALUE := 0.0;
   STATUS[949].TRIGVALUE := 0.0;
   STATUS[949].EXT.AlarmWarnUnAck := FALSE;
   STATUS[949].EXT.AckRequired := FALSE;
   STATUS[949].EXT.Maintanence := FALSE;
   STATUS[949].EXT.Operation := FALSE;
   STATUS[949].EXT.Forced := FALSE;
   STATUS[949].EXT.BIT29 := FALSE;
   STATUS[949].EXT.BIT30 := FALSE;
   STATUS[949].EXT.BIT31 := FALSE;
   STATUS[949].EXT.ModeBit1 := FALSE;
   STATUS[949].EXT.ModeBit2 := FALSE;
   STATUS[949].EXT.ModeBit3 := FALSE;
   STATUS[949].EXT.BIT19 := FALSE;
   STATUS[949].EXT.BIT20 := FALSE;
   STATUS[949].EXT.AlarmSuppressed := FALSE;
   STATUS[949].EXT.AlarmPrsent := FALSE;
   STATUS[949].EXT.AlarmFailUnAck := FALSE;
   STATUS[949].Status := 0;
   STATUS[949].TimeStamp := 16#0000;
   STATUS[950].VALUE := 0.0;
   STATUS[950].TRIGVALUE := 0.0;
   STATUS[950].EXT.AlarmWarnUnAck := FALSE;
   STATUS[950].EXT.AckRequired := FALSE;
   STATUS[950].EXT.Maintanence := FALSE;
   STATUS[950].EXT.Operation := FALSE;
   STATUS[950].EXT.Forced := FALSE;
   STATUS[950].EXT.BIT29 := FALSE;
   STATUS[950].EXT.BIT30 := FALSE;
   STATUS[950].EXT.BIT31 := FALSE;
   STATUS[950].EXT.ModeBit1 := FALSE;
   STATUS[950].EXT.ModeBit2 := FALSE;
   STATUS[950].EXT.ModeBit3 := FALSE;
   STATUS[950].EXT.BIT19 := FALSE;
   STATUS[950].EXT.BIT20 := FALSE;
   STATUS[950].EXT.AlarmSuppressed := FALSE;
   STATUS[950].EXT.AlarmPrsent := FALSE;
   STATUS[950].EXT.AlarmFailUnAck := FALSE;
   STATUS[950].Status := 0;
   STATUS[950].TimeStamp := 16#0000;
   STATUS[951].VALUE := 0.0;
   STATUS[951].TRIGVALUE := 0.0;
   STATUS[951].EXT.AlarmWarnUnAck := FALSE;
   STATUS[951].EXT.AckRequired := FALSE;
   STATUS[951].EXT.Maintanence := FALSE;
   STATUS[951].EXT.Operation := FALSE;
   STATUS[951].EXT.Forced := FALSE;
   STATUS[951].EXT.BIT29 := FALSE;
   STATUS[951].EXT.BIT30 := FALSE;
   STATUS[951].EXT.BIT31 := FALSE;
   STATUS[951].EXT.ModeBit1 := FALSE;
   STATUS[951].EXT.ModeBit2 := FALSE;
   STATUS[951].EXT.ModeBit3 := FALSE;
   STATUS[951].EXT.BIT19 := FALSE;
   STATUS[951].EXT.BIT20 := FALSE;
   STATUS[951].EXT.AlarmSuppressed := FALSE;
   STATUS[951].EXT.AlarmPrsent := FALSE;
   STATUS[951].EXT.AlarmFailUnAck := FALSE;
   STATUS[951].Status := 0;
   STATUS[951].TimeStamp := 16#0000;
   STATUS[952].VALUE := 0.0;
   STATUS[952].TRIGVALUE := 0.0;
   STATUS[952].EXT.AlarmWarnUnAck := FALSE;
   STATUS[952].EXT.AckRequired := FALSE;
   STATUS[952].EXT.Maintanence := FALSE;
   STATUS[952].EXT.Operation := FALSE;
   STATUS[952].EXT.Forced := FALSE;
   STATUS[952].EXT.BIT29 := FALSE;
   STATUS[952].EXT.BIT30 := FALSE;
   STATUS[952].EXT.BIT31 := FALSE;
   STATUS[952].EXT.ModeBit1 := FALSE;
   STATUS[952].EXT.ModeBit2 := FALSE;
   STATUS[952].EXT.ModeBit3 := FALSE;
   STATUS[952].EXT.BIT19 := FALSE;
   STATUS[952].EXT.BIT20 := FALSE;
   STATUS[952].EXT.AlarmSuppressed := FALSE;
   STATUS[952].EXT.AlarmPrsent := FALSE;
   STATUS[952].EXT.AlarmFailUnAck := FALSE;
   STATUS[952].Status := 0;
   STATUS[952].TimeStamp := 16#0000;
   STATUS[953].VALUE := 0.0;
   STATUS[953].TRIGVALUE := 0.0;
   STATUS[953].EXT.AlarmWarnUnAck := FALSE;
   STATUS[953].EXT.AckRequired := FALSE;
   STATUS[953].EXT.Maintanence := FALSE;
   STATUS[953].EXT.Operation := FALSE;
   STATUS[953].EXT.Forced := FALSE;
   STATUS[953].EXT.BIT29 := FALSE;
   STATUS[953].EXT.BIT30 := FALSE;
   STATUS[953].EXT.BIT31 := FALSE;
   STATUS[953].EXT.ModeBit1 := FALSE;
   STATUS[953].EXT.ModeBit2 := FALSE;
   STATUS[953].EXT.ModeBit3 := FALSE;
   STATUS[953].EXT.BIT19 := FALSE;
   STATUS[953].EXT.BIT20 := FALSE;
   STATUS[953].EXT.AlarmSuppressed := FALSE;
   STATUS[953].EXT.AlarmPrsent := FALSE;
   STATUS[953].EXT.AlarmFailUnAck := FALSE;
   STATUS[953].Status := 0;
   STATUS[953].TimeStamp := 16#0000;
   STATUS[954].VALUE := 0.0;
   STATUS[954].TRIGVALUE := 0.0;
   STATUS[954].EXT.AlarmWarnUnAck := FALSE;
   STATUS[954].EXT.AckRequired := FALSE;
   STATUS[954].EXT.Maintanence := FALSE;
   STATUS[954].EXT.Operation := FALSE;
   STATUS[954].EXT.Forced := FALSE;
   STATUS[954].EXT.BIT29 := FALSE;
   STATUS[954].EXT.BIT30 := FALSE;
   STATUS[954].EXT.BIT31 := FALSE;
   STATUS[954].EXT.ModeBit1 := FALSE;
   STATUS[954].EXT.ModeBit2 := FALSE;
   STATUS[954].EXT.ModeBit3 := FALSE;
   STATUS[954].EXT.BIT19 := FALSE;
   STATUS[954].EXT.BIT20 := FALSE;
   STATUS[954].EXT.AlarmSuppressed := FALSE;
   STATUS[954].EXT.AlarmPrsent := FALSE;
   STATUS[954].EXT.AlarmFailUnAck := FALSE;
   STATUS[954].Status := 0;
   STATUS[954].TimeStamp := 16#0000;
   STATUS[955].VALUE := 0.0;
   STATUS[955].TRIGVALUE := 0.0;
   STATUS[955].EXT.AlarmWarnUnAck := FALSE;
   STATUS[955].EXT.AckRequired := FALSE;
   STATUS[955].EXT.Maintanence := FALSE;
   STATUS[955].EXT.Operation := FALSE;
   STATUS[955].EXT.Forced := FALSE;
   STATUS[955].EXT.BIT29 := FALSE;
   STATUS[955].EXT.BIT30 := FALSE;
   STATUS[955].EXT.BIT31 := FALSE;
   STATUS[955].EXT.ModeBit1 := FALSE;
   STATUS[955].EXT.ModeBit2 := FALSE;
   STATUS[955].EXT.ModeBit3 := FALSE;
   STATUS[955].EXT.BIT19 := FALSE;
   STATUS[955].EXT.BIT20 := FALSE;
   STATUS[955].EXT.AlarmSuppressed := FALSE;
   STATUS[955].EXT.AlarmPrsent := FALSE;
   STATUS[955].EXT.AlarmFailUnAck := FALSE;
   STATUS[955].Status := 0;
   STATUS[955].TimeStamp := 16#0000;
   STATUS[956].VALUE := 0.0;
   STATUS[956].TRIGVALUE := 0.0;
   STATUS[956].EXT.AlarmWarnUnAck := FALSE;
   STATUS[956].EXT.AckRequired := FALSE;
   STATUS[956].EXT.Maintanence := FALSE;
   STATUS[956].EXT.Operation := FALSE;
   STATUS[956].EXT.Forced := FALSE;
   STATUS[956].EXT.BIT29 := FALSE;
   STATUS[956].EXT.BIT30 := FALSE;
   STATUS[956].EXT.BIT31 := FALSE;
   STATUS[956].EXT.ModeBit1 := FALSE;
   STATUS[956].EXT.ModeBit2 := FALSE;
   STATUS[956].EXT.ModeBit3 := FALSE;
   STATUS[956].EXT.BIT19 := FALSE;
   STATUS[956].EXT.BIT20 := FALSE;
   STATUS[956].EXT.AlarmSuppressed := FALSE;
   STATUS[956].EXT.AlarmPrsent := FALSE;
   STATUS[956].EXT.AlarmFailUnAck := FALSE;
   STATUS[956].Status := 0;
   STATUS[956].TimeStamp := 16#0000;
   STATUS[957].VALUE := 0.0;
   STATUS[957].TRIGVALUE := 0.0;
   STATUS[957].EXT.AlarmWarnUnAck := FALSE;
   STATUS[957].EXT.AckRequired := FALSE;
   STATUS[957].EXT.Maintanence := FALSE;
   STATUS[957].EXT.Operation := FALSE;
   STATUS[957].EXT.Forced := FALSE;
   STATUS[957].EXT.BIT29 := FALSE;
   STATUS[957].EXT.BIT30 := FALSE;
   STATUS[957].EXT.BIT31 := FALSE;
   STATUS[957].EXT.ModeBit1 := FALSE;
   STATUS[957].EXT.ModeBit2 := FALSE;
   STATUS[957].EXT.ModeBit3 := FALSE;
   STATUS[957].EXT.BIT19 := FALSE;
   STATUS[957].EXT.BIT20 := FALSE;
   STATUS[957].EXT.AlarmSuppressed := FALSE;
   STATUS[957].EXT.AlarmPrsent := FALSE;
   STATUS[957].EXT.AlarmFailUnAck := FALSE;
   STATUS[957].Status := 0;
   STATUS[957].TimeStamp := 16#0000;
   STATUS[958].VALUE := 0.0;
   STATUS[958].TRIGVALUE := 0.0;
   STATUS[958].EXT.AlarmWarnUnAck := FALSE;
   STATUS[958].EXT.AckRequired := FALSE;
   STATUS[958].EXT.Maintanence := FALSE;
   STATUS[958].EXT.Operation := FALSE;
   STATUS[958].EXT.Forced := FALSE;
   STATUS[958].EXT.BIT29 := FALSE;
   STATUS[958].EXT.BIT30 := FALSE;
   STATUS[958].EXT.BIT31 := FALSE;
   STATUS[958].EXT.ModeBit1 := FALSE;
   STATUS[958].EXT.ModeBit2 := FALSE;
   STATUS[958].EXT.ModeBit3 := FALSE;
   STATUS[958].EXT.BIT19 := FALSE;
   STATUS[958].EXT.BIT20 := FALSE;
   STATUS[958].EXT.AlarmSuppressed := FALSE;
   STATUS[958].EXT.AlarmPrsent := FALSE;
   STATUS[958].EXT.AlarmFailUnAck := FALSE;
   STATUS[958].Status := 0;
   STATUS[958].TimeStamp := 16#0000;
   STATUS[959].VALUE := 0.0;
   STATUS[959].TRIGVALUE := 0.0;
   STATUS[959].EXT.AlarmWarnUnAck := FALSE;
   STATUS[959].EXT.AckRequired := FALSE;
   STATUS[959].EXT.Maintanence := FALSE;
   STATUS[959].EXT.Operation := FALSE;
   STATUS[959].EXT.Forced := FALSE;
   STATUS[959].EXT.BIT29 := FALSE;
   STATUS[959].EXT.BIT30 := FALSE;
   STATUS[959].EXT.BIT31 := FALSE;
   STATUS[959].EXT.ModeBit1 := FALSE;
   STATUS[959].EXT.ModeBit2 := FALSE;
   STATUS[959].EXT.ModeBit3 := FALSE;
   STATUS[959].EXT.BIT19 := FALSE;
   STATUS[959].EXT.BIT20 := FALSE;
   STATUS[959].EXT.AlarmSuppressed := FALSE;
   STATUS[959].EXT.AlarmPrsent := FALSE;
   STATUS[959].EXT.AlarmFailUnAck := FALSE;
   STATUS[959].Status := 0;
   STATUS[959].TimeStamp := 16#0000;
   STATUS[960].VALUE := 0.0;
   STATUS[960].TRIGVALUE := 0.0;
   STATUS[960].EXT.AlarmWarnUnAck := FALSE;
   STATUS[960].EXT.AckRequired := FALSE;
   STATUS[960].EXT.Maintanence := FALSE;
   STATUS[960].EXT.Operation := FALSE;
   STATUS[960].EXT.Forced := FALSE;
   STATUS[960].EXT.BIT29 := FALSE;
   STATUS[960].EXT.BIT30 := FALSE;
   STATUS[960].EXT.BIT31 := FALSE;
   STATUS[960].EXT.ModeBit1 := FALSE;
   STATUS[960].EXT.ModeBit2 := FALSE;
   STATUS[960].EXT.ModeBit3 := FALSE;
   STATUS[960].EXT.BIT19 := FALSE;
   STATUS[960].EXT.BIT20 := FALSE;
   STATUS[960].EXT.AlarmSuppressed := FALSE;
   STATUS[960].EXT.AlarmPrsent := FALSE;
   STATUS[960].EXT.AlarmFailUnAck := FALSE;
   STATUS[960].Status := 0;
   STATUS[960].TimeStamp := 16#0000;
   STATUS[961].VALUE := 0.0;
   STATUS[961].TRIGVALUE := 0.0;
   STATUS[961].EXT.AlarmWarnUnAck := FALSE;
   STATUS[961].EXT.AckRequired := FALSE;
   STATUS[961].EXT.Maintanence := FALSE;
   STATUS[961].EXT.Operation := FALSE;
   STATUS[961].EXT.Forced := FALSE;
   STATUS[961].EXT.BIT29 := FALSE;
   STATUS[961].EXT.BIT30 := FALSE;
   STATUS[961].EXT.BIT31 := FALSE;
   STATUS[961].EXT.ModeBit1 := FALSE;
   STATUS[961].EXT.ModeBit2 := FALSE;
   STATUS[961].EXT.ModeBit3 := FALSE;
   STATUS[961].EXT.BIT19 := FALSE;
   STATUS[961].EXT.BIT20 := FALSE;
   STATUS[961].EXT.AlarmSuppressed := FALSE;
   STATUS[961].EXT.AlarmPrsent := FALSE;
   STATUS[961].EXT.AlarmFailUnAck := FALSE;
   STATUS[961].Status := 0;
   STATUS[961].TimeStamp := 16#0000;
   STATUS[962].VALUE := 0.0;
   STATUS[962].TRIGVALUE := 0.0;
   STATUS[962].EXT.AlarmWarnUnAck := FALSE;
   STATUS[962].EXT.AckRequired := FALSE;
   STATUS[962].EXT.Maintanence := FALSE;
   STATUS[962].EXT.Operation := FALSE;
   STATUS[962].EXT.Forced := FALSE;
   STATUS[962].EXT.BIT29 := FALSE;
   STATUS[962].EXT.BIT30 := FALSE;
   STATUS[962].EXT.BIT31 := FALSE;
   STATUS[962].EXT.ModeBit1 := FALSE;
   STATUS[962].EXT.ModeBit2 := FALSE;
   STATUS[962].EXT.ModeBit3 := FALSE;
   STATUS[962].EXT.BIT19 := FALSE;
   STATUS[962].EXT.BIT20 := FALSE;
   STATUS[962].EXT.AlarmSuppressed := FALSE;
   STATUS[962].EXT.AlarmPrsent := FALSE;
   STATUS[962].EXT.AlarmFailUnAck := FALSE;
   STATUS[962].Status := 0;
   STATUS[962].TimeStamp := 16#0000;
   STATUS[963].VALUE := 0.0;
   STATUS[963].TRIGVALUE := 0.0;
   STATUS[963].EXT.AlarmWarnUnAck := FALSE;
   STATUS[963].EXT.AckRequired := FALSE;
   STATUS[963].EXT.Maintanence := FALSE;
   STATUS[963].EXT.Operation := FALSE;
   STATUS[963].EXT.Forced := FALSE;
   STATUS[963].EXT.BIT29 := FALSE;
   STATUS[963].EXT.BIT30 := FALSE;
   STATUS[963].EXT.BIT31 := FALSE;
   STATUS[963].EXT.ModeBit1 := FALSE;
   STATUS[963].EXT.ModeBit2 := FALSE;
   STATUS[963].EXT.ModeBit3 := FALSE;
   STATUS[963].EXT.BIT19 := FALSE;
   STATUS[963].EXT.BIT20 := FALSE;
   STATUS[963].EXT.AlarmSuppressed := FALSE;
   STATUS[963].EXT.AlarmPrsent := FALSE;
   STATUS[963].EXT.AlarmFailUnAck := FALSE;
   STATUS[963].Status := 0;
   STATUS[963].TimeStamp := 16#0000;
   STATUS[964].VALUE := 0.0;
   STATUS[964].TRIGVALUE := 0.0;
   STATUS[964].EXT.AlarmWarnUnAck := FALSE;
   STATUS[964].EXT.AckRequired := FALSE;
   STATUS[964].EXT.Maintanence := FALSE;
   STATUS[964].EXT.Operation := FALSE;
   STATUS[964].EXT.Forced := FALSE;
   STATUS[964].EXT.BIT29 := FALSE;
   STATUS[964].EXT.BIT30 := FALSE;
   STATUS[964].EXT.BIT31 := FALSE;
   STATUS[964].EXT.ModeBit1 := FALSE;
   STATUS[964].EXT.ModeBit2 := FALSE;
   STATUS[964].EXT.ModeBit3 := FALSE;
   STATUS[964].EXT.BIT19 := FALSE;
   STATUS[964].EXT.BIT20 := FALSE;
   STATUS[964].EXT.AlarmSuppressed := FALSE;
   STATUS[964].EXT.AlarmPrsent := FALSE;
   STATUS[964].EXT.AlarmFailUnAck := FALSE;
   STATUS[964].Status := 0;
   STATUS[964].TimeStamp := 16#0000;
   STATUS[965].VALUE := 0.0;
   STATUS[965].TRIGVALUE := 0.0;
   STATUS[965].EXT.AlarmWarnUnAck := FALSE;
   STATUS[965].EXT.AckRequired := FALSE;
   STATUS[965].EXT.Maintanence := FALSE;
   STATUS[965].EXT.Operation := FALSE;
   STATUS[965].EXT.Forced := FALSE;
   STATUS[965].EXT.BIT29 := FALSE;
   STATUS[965].EXT.BIT30 := FALSE;
   STATUS[965].EXT.BIT31 := FALSE;
   STATUS[965].EXT.ModeBit1 := FALSE;
   STATUS[965].EXT.ModeBit2 := FALSE;
   STATUS[965].EXT.ModeBit3 := FALSE;
   STATUS[965].EXT.BIT19 := FALSE;
   STATUS[965].EXT.BIT20 := FALSE;
   STATUS[965].EXT.AlarmSuppressed := FALSE;
   STATUS[965].EXT.AlarmPrsent := FALSE;
   STATUS[965].EXT.AlarmFailUnAck := FALSE;
   STATUS[965].Status := 0;
   STATUS[965].TimeStamp := 16#0000;
   STATUS[966].VALUE := 0.0;
   STATUS[966].TRIGVALUE := 0.0;
   STATUS[966].EXT.AlarmWarnUnAck := FALSE;
   STATUS[966].EXT.AckRequired := FALSE;
   STATUS[966].EXT.Maintanence := FALSE;
   STATUS[966].EXT.Operation := FALSE;
   STATUS[966].EXT.Forced := FALSE;
   STATUS[966].EXT.BIT29 := FALSE;
   STATUS[966].EXT.BIT30 := FALSE;
   STATUS[966].EXT.BIT31 := FALSE;
   STATUS[966].EXT.ModeBit1 := FALSE;
   STATUS[966].EXT.ModeBit2 := FALSE;
   STATUS[966].EXT.ModeBit3 := FALSE;
   STATUS[966].EXT.BIT19 := FALSE;
   STATUS[966].EXT.BIT20 := FALSE;
   STATUS[966].EXT.AlarmSuppressed := FALSE;
   STATUS[966].EXT.AlarmPrsent := FALSE;
   STATUS[966].EXT.AlarmFailUnAck := FALSE;
   STATUS[966].Status := 0;
   STATUS[966].TimeStamp := 16#0000;
   STATUS[967].VALUE := 0.0;
   STATUS[967].TRIGVALUE := 0.0;
   STATUS[967].EXT.AlarmWarnUnAck := FALSE;
   STATUS[967].EXT.AckRequired := FALSE;
   STATUS[967].EXT.Maintanence := FALSE;
   STATUS[967].EXT.Operation := FALSE;
   STATUS[967].EXT.Forced := FALSE;
   STATUS[967].EXT.BIT29 := FALSE;
   STATUS[967].EXT.BIT30 := FALSE;
   STATUS[967].EXT.BIT31 := FALSE;
   STATUS[967].EXT.ModeBit1 := FALSE;
   STATUS[967].EXT.ModeBit2 := FALSE;
   STATUS[967].EXT.ModeBit3 := FALSE;
   STATUS[967].EXT.BIT19 := FALSE;
   STATUS[967].EXT.BIT20 := FALSE;
   STATUS[967].EXT.AlarmSuppressed := FALSE;
   STATUS[967].EXT.AlarmPrsent := FALSE;
   STATUS[967].EXT.AlarmFailUnAck := FALSE;
   STATUS[967].Status := 0;
   STATUS[967].TimeStamp := 16#0000;
   STATUS[968].VALUE := 0.0;
   STATUS[968].TRIGVALUE := 0.0;
   STATUS[968].EXT.AlarmWarnUnAck := FALSE;
   STATUS[968].EXT.AckRequired := FALSE;
   STATUS[968].EXT.Maintanence := FALSE;
   STATUS[968].EXT.Operation := FALSE;
   STATUS[968].EXT.Forced := FALSE;
   STATUS[968].EXT.BIT29 := FALSE;
   STATUS[968].EXT.BIT30 := FALSE;
   STATUS[968].EXT.BIT31 := FALSE;
   STATUS[968].EXT.ModeBit1 := FALSE;
   STATUS[968].EXT.ModeBit2 := FALSE;
   STATUS[968].EXT.ModeBit3 := FALSE;
   STATUS[968].EXT.BIT19 := FALSE;
   STATUS[968].EXT.BIT20 := FALSE;
   STATUS[968].EXT.AlarmSuppressed := FALSE;
   STATUS[968].EXT.AlarmPrsent := FALSE;
   STATUS[968].EXT.AlarmFailUnAck := FALSE;
   STATUS[968].Status := 0;
   STATUS[968].TimeStamp := 16#0000;
   STATUS[969].VALUE := 0.0;
   STATUS[969].TRIGVALUE := 0.0;
   STATUS[969].EXT.AlarmWarnUnAck := FALSE;
   STATUS[969].EXT.AckRequired := FALSE;
   STATUS[969].EXT.Maintanence := FALSE;
   STATUS[969].EXT.Operation := FALSE;
   STATUS[969].EXT.Forced := FALSE;
   STATUS[969].EXT.BIT29 := FALSE;
   STATUS[969].EXT.BIT30 := FALSE;
   STATUS[969].EXT.BIT31 := FALSE;
   STATUS[969].EXT.ModeBit1 := FALSE;
   STATUS[969].EXT.ModeBit2 := FALSE;
   STATUS[969].EXT.ModeBit3 := FALSE;
   STATUS[969].EXT.BIT19 := FALSE;
   STATUS[969].EXT.BIT20 := FALSE;
   STATUS[969].EXT.AlarmSuppressed := FALSE;
   STATUS[969].EXT.AlarmPrsent := FALSE;
   STATUS[969].EXT.AlarmFailUnAck := FALSE;
   STATUS[969].Status := 0;
   STATUS[969].TimeStamp := 16#0000;
   STATUS[970].VALUE := 0.0;
   STATUS[970].TRIGVALUE := 0.0;
   STATUS[970].EXT.AlarmWarnUnAck := FALSE;
   STATUS[970].EXT.AckRequired := FALSE;
   STATUS[970].EXT.Maintanence := FALSE;
   STATUS[970].EXT.Operation := FALSE;
   STATUS[970].EXT.Forced := FALSE;
   STATUS[970].EXT.BIT29 := FALSE;
   STATUS[970].EXT.BIT30 := FALSE;
   STATUS[970].EXT.BIT31 := FALSE;
   STATUS[970].EXT.ModeBit1 := FALSE;
   STATUS[970].EXT.ModeBit2 := FALSE;
   STATUS[970].EXT.ModeBit3 := FALSE;
   STATUS[970].EXT.BIT19 := FALSE;
   STATUS[970].EXT.BIT20 := FALSE;
   STATUS[970].EXT.AlarmSuppressed := FALSE;
   STATUS[970].EXT.AlarmPrsent := FALSE;
   STATUS[970].EXT.AlarmFailUnAck := FALSE;
   STATUS[970].Status := 0;
   STATUS[970].TimeStamp := 16#0000;
   STATUS[971].VALUE := 0.0;
   STATUS[971].TRIGVALUE := 0.0;
   STATUS[971].EXT.AlarmWarnUnAck := FALSE;
   STATUS[971].EXT.AckRequired := FALSE;
   STATUS[971].EXT.Maintanence := FALSE;
   STATUS[971].EXT.Operation := FALSE;
   STATUS[971].EXT.Forced := FALSE;
   STATUS[971].EXT.BIT29 := FALSE;
   STATUS[971].EXT.BIT30 := FALSE;
   STATUS[971].EXT.BIT31 := FALSE;
   STATUS[971].EXT.ModeBit1 := FALSE;
   STATUS[971].EXT.ModeBit2 := FALSE;
   STATUS[971].EXT.ModeBit3 := FALSE;
   STATUS[971].EXT.BIT19 := FALSE;
   STATUS[971].EXT.BIT20 := FALSE;
   STATUS[971].EXT.AlarmSuppressed := FALSE;
   STATUS[971].EXT.AlarmPrsent := FALSE;
   STATUS[971].EXT.AlarmFailUnAck := FALSE;
   STATUS[971].Status := 0;
   STATUS[971].TimeStamp := 16#0000;
   STATUS[972].VALUE := 0.0;
   STATUS[972].TRIGVALUE := 0.0;
   STATUS[972].EXT.AlarmWarnUnAck := FALSE;
   STATUS[972].EXT.AckRequired := FALSE;
   STATUS[972].EXT.Maintanence := FALSE;
   STATUS[972].EXT.Operation := FALSE;
   STATUS[972].EXT.Forced := FALSE;
   STATUS[972].EXT.BIT29 := FALSE;
   STATUS[972].EXT.BIT30 := FALSE;
   STATUS[972].EXT.BIT31 := FALSE;
   STATUS[972].EXT.ModeBit1 := FALSE;
   STATUS[972].EXT.ModeBit2 := FALSE;
   STATUS[972].EXT.ModeBit3 := FALSE;
   STATUS[972].EXT.BIT19 := FALSE;
   STATUS[972].EXT.BIT20 := FALSE;
   STATUS[972].EXT.AlarmSuppressed := FALSE;
   STATUS[972].EXT.AlarmPrsent := FALSE;
   STATUS[972].EXT.AlarmFailUnAck := FALSE;
   STATUS[972].Status := 0;
   STATUS[972].TimeStamp := 16#0000;
   STATUS[973].VALUE := 0.0;
   STATUS[973].TRIGVALUE := 0.0;
   STATUS[973].EXT.AlarmWarnUnAck := FALSE;
   STATUS[973].EXT.AckRequired := FALSE;
   STATUS[973].EXT.Maintanence := FALSE;
   STATUS[973].EXT.Operation := FALSE;
   STATUS[973].EXT.Forced := FALSE;
   STATUS[973].EXT.BIT29 := FALSE;
   STATUS[973].EXT.BIT30 := FALSE;
   STATUS[973].EXT.BIT31 := FALSE;
   STATUS[973].EXT.ModeBit1 := FALSE;
   STATUS[973].EXT.ModeBit2 := FALSE;
   STATUS[973].EXT.ModeBit3 := FALSE;
   STATUS[973].EXT.BIT19 := FALSE;
   STATUS[973].EXT.BIT20 := FALSE;
   STATUS[973].EXT.AlarmSuppressed := FALSE;
   STATUS[973].EXT.AlarmPrsent := FALSE;
   STATUS[973].EXT.AlarmFailUnAck := FALSE;
   STATUS[973].Status := 0;
   STATUS[973].TimeStamp := 16#0000;
   STATUS[974].VALUE := 0.0;
   STATUS[974].TRIGVALUE := 0.0;
   STATUS[974].EXT.AlarmWarnUnAck := FALSE;
   STATUS[974].EXT.AckRequired := FALSE;
   STATUS[974].EXT.Maintanence := FALSE;
   STATUS[974].EXT.Operation := FALSE;
   STATUS[974].EXT.Forced := FALSE;
   STATUS[974].EXT.BIT29 := FALSE;
   STATUS[974].EXT.BIT30 := FALSE;
   STATUS[974].EXT.BIT31 := FALSE;
   STATUS[974].EXT.ModeBit1 := FALSE;
   STATUS[974].EXT.ModeBit2 := FALSE;
   STATUS[974].EXT.ModeBit3 := FALSE;
   STATUS[974].EXT.BIT19 := FALSE;
   STATUS[974].EXT.BIT20 := FALSE;
   STATUS[974].EXT.AlarmSuppressed := FALSE;
   STATUS[974].EXT.AlarmPrsent := FALSE;
   STATUS[974].EXT.AlarmFailUnAck := FALSE;
   STATUS[974].Status := 0;
   STATUS[974].TimeStamp := 16#0000;
   STATUS[975].VALUE := 0.0;
   STATUS[975].TRIGVALUE := 0.0;
   STATUS[975].EXT.AlarmWarnUnAck := FALSE;
   STATUS[975].EXT.AckRequired := FALSE;
   STATUS[975].EXT.Maintanence := FALSE;
   STATUS[975].EXT.Operation := FALSE;
   STATUS[975].EXT.Forced := FALSE;
   STATUS[975].EXT.BIT29 := FALSE;
   STATUS[975].EXT.BIT30 := FALSE;
   STATUS[975].EXT.BIT31 := FALSE;
   STATUS[975].EXT.ModeBit1 := FALSE;
   STATUS[975].EXT.ModeBit2 := FALSE;
   STATUS[975].EXT.ModeBit3 := FALSE;
   STATUS[975].EXT.BIT19 := FALSE;
   STATUS[975].EXT.BIT20 := FALSE;
   STATUS[975].EXT.AlarmSuppressed := FALSE;
   STATUS[975].EXT.AlarmPrsent := FALSE;
   STATUS[975].EXT.AlarmFailUnAck := FALSE;
   STATUS[975].Status := 0;
   STATUS[975].TimeStamp := 16#0000;
   STATUS[976].VALUE := 0.0;
   STATUS[976].TRIGVALUE := 0.0;
   STATUS[976].EXT.AlarmWarnUnAck := FALSE;
   STATUS[976].EXT.AckRequired := FALSE;
   STATUS[976].EXT.Maintanence := FALSE;
   STATUS[976].EXT.Operation := FALSE;
   STATUS[976].EXT.Forced := FALSE;
   STATUS[976].EXT.BIT29 := FALSE;
   STATUS[976].EXT.BIT30 := FALSE;
   STATUS[976].EXT.BIT31 := FALSE;
   STATUS[976].EXT.ModeBit1 := FALSE;
   STATUS[976].EXT.ModeBit2 := FALSE;
   STATUS[976].EXT.ModeBit3 := FALSE;
   STATUS[976].EXT.BIT19 := FALSE;
   STATUS[976].EXT.BIT20 := FALSE;
   STATUS[976].EXT.AlarmSuppressed := FALSE;
   STATUS[976].EXT.AlarmPrsent := FALSE;
   STATUS[976].EXT.AlarmFailUnAck := FALSE;
   STATUS[976].Status := 0;
   STATUS[976].TimeStamp := 16#0000;
   STATUS[977].VALUE := 0.0;
   STATUS[977].TRIGVALUE := 0.0;
   STATUS[977].EXT.AlarmWarnUnAck := FALSE;
   STATUS[977].EXT.AckRequired := FALSE;
   STATUS[977].EXT.Maintanence := FALSE;
   STATUS[977].EXT.Operation := FALSE;
   STATUS[977].EXT.Forced := FALSE;
   STATUS[977].EXT.BIT29 := FALSE;
   STATUS[977].EXT.BIT30 := FALSE;
   STATUS[977].EXT.BIT31 := FALSE;
   STATUS[977].EXT.ModeBit1 := FALSE;
   STATUS[977].EXT.ModeBit2 := FALSE;
   STATUS[977].EXT.ModeBit3 := FALSE;
   STATUS[977].EXT.BIT19 := FALSE;
   STATUS[977].EXT.BIT20 := FALSE;
   STATUS[977].EXT.AlarmSuppressed := FALSE;
   STATUS[977].EXT.AlarmPrsent := FALSE;
   STATUS[977].EXT.AlarmFailUnAck := FALSE;
   STATUS[977].Status := 0;
   STATUS[977].TimeStamp := 16#0000;
   STATUS[978].VALUE := 0.0;
   STATUS[978].TRIGVALUE := 0.0;
   STATUS[978].EXT.AlarmWarnUnAck := FALSE;
   STATUS[978].EXT.AckRequired := FALSE;
   STATUS[978].EXT.Maintanence := FALSE;
   STATUS[978].EXT.Operation := FALSE;
   STATUS[978].EXT.Forced := FALSE;
   STATUS[978].EXT.BIT29 := FALSE;
   STATUS[978].EXT.BIT30 := FALSE;
   STATUS[978].EXT.BIT31 := FALSE;
   STATUS[978].EXT.ModeBit1 := FALSE;
   STATUS[978].EXT.ModeBit2 := FALSE;
   STATUS[978].EXT.ModeBit3 := FALSE;
   STATUS[978].EXT.BIT19 := FALSE;
   STATUS[978].EXT.BIT20 := FALSE;
   STATUS[978].EXT.AlarmSuppressed := FALSE;
   STATUS[978].EXT.AlarmPrsent := FALSE;
   STATUS[978].EXT.AlarmFailUnAck := FALSE;
   STATUS[978].Status := 0;
   STATUS[978].TimeStamp := 16#0000;
   STATUS[979].VALUE := 0.0;
   STATUS[979].TRIGVALUE := 0.0;
   STATUS[979].EXT.AlarmWarnUnAck := FALSE;
   STATUS[979].EXT.AckRequired := FALSE;
   STATUS[979].EXT.Maintanence := FALSE;
   STATUS[979].EXT.Operation := FALSE;
   STATUS[979].EXT.Forced := FALSE;
   STATUS[979].EXT.BIT29 := FALSE;
   STATUS[979].EXT.BIT30 := FALSE;
   STATUS[979].EXT.BIT31 := FALSE;
   STATUS[979].EXT.ModeBit1 := FALSE;
   STATUS[979].EXT.ModeBit2 := FALSE;
   STATUS[979].EXT.ModeBit3 := FALSE;
   STATUS[979].EXT.BIT19 := FALSE;
   STATUS[979].EXT.BIT20 := FALSE;
   STATUS[979].EXT.AlarmSuppressed := FALSE;
   STATUS[979].EXT.AlarmPrsent := FALSE;
   STATUS[979].EXT.AlarmFailUnAck := FALSE;
   STATUS[979].Status := 0;
   STATUS[979].TimeStamp := 16#0000;
   STATUS[980].VALUE := 0.0;
   STATUS[980].TRIGVALUE := 0.0;
   STATUS[980].EXT.AlarmWarnUnAck := FALSE;
   STATUS[980].EXT.AckRequired := FALSE;
   STATUS[980].EXT.Maintanence := FALSE;
   STATUS[980].EXT.Operation := FALSE;
   STATUS[980].EXT.Forced := FALSE;
   STATUS[980].EXT.BIT29 := FALSE;
   STATUS[980].EXT.BIT30 := FALSE;
   STATUS[980].EXT.BIT31 := FALSE;
   STATUS[980].EXT.ModeBit1 := FALSE;
   STATUS[980].EXT.ModeBit2 := FALSE;
   STATUS[980].EXT.ModeBit3 := FALSE;
   STATUS[980].EXT.BIT19 := FALSE;
   STATUS[980].EXT.BIT20 := FALSE;
   STATUS[980].EXT.AlarmSuppressed := FALSE;
   STATUS[980].EXT.AlarmPrsent := FALSE;
   STATUS[980].EXT.AlarmFailUnAck := FALSE;
   STATUS[980].Status := 0;
   STATUS[980].TimeStamp := 16#0000;
   STATUS[981].VALUE := 0.0;
   STATUS[981].TRIGVALUE := 0.0;
   STATUS[981].EXT.AlarmWarnUnAck := FALSE;
   STATUS[981].EXT.AckRequired := FALSE;
   STATUS[981].EXT.Maintanence := FALSE;
   STATUS[981].EXT.Operation := FALSE;
   STATUS[981].EXT.Forced := FALSE;
   STATUS[981].EXT.BIT29 := FALSE;
   STATUS[981].EXT.BIT30 := FALSE;
   STATUS[981].EXT.BIT31 := FALSE;
   STATUS[981].EXT.ModeBit1 := FALSE;
   STATUS[981].EXT.ModeBit2 := FALSE;
   STATUS[981].EXT.ModeBit3 := FALSE;
   STATUS[981].EXT.BIT19 := FALSE;
   STATUS[981].EXT.BIT20 := FALSE;
   STATUS[981].EXT.AlarmSuppressed := FALSE;
   STATUS[981].EXT.AlarmPrsent := FALSE;
   STATUS[981].EXT.AlarmFailUnAck := FALSE;
   STATUS[981].Status := 0;
   STATUS[981].TimeStamp := 16#0000;
   STATUS[982].VALUE := 0.0;
   STATUS[982].TRIGVALUE := 0.0;
   STATUS[982].EXT.AlarmWarnUnAck := FALSE;
   STATUS[982].EXT.AckRequired := FALSE;
   STATUS[982].EXT.Maintanence := FALSE;
   STATUS[982].EXT.Operation := FALSE;
   STATUS[982].EXT.Forced := FALSE;
   STATUS[982].EXT.BIT29 := FALSE;
   STATUS[982].EXT.BIT30 := FALSE;
   STATUS[982].EXT.BIT31 := FALSE;
   STATUS[982].EXT.ModeBit1 := FALSE;
   STATUS[982].EXT.ModeBit2 := FALSE;
   STATUS[982].EXT.ModeBit3 := FALSE;
   STATUS[982].EXT.BIT19 := FALSE;
   STATUS[982].EXT.BIT20 := FALSE;
   STATUS[982].EXT.AlarmSuppressed := FALSE;
   STATUS[982].EXT.AlarmPrsent := FALSE;
   STATUS[982].EXT.AlarmFailUnAck := FALSE;
   STATUS[982].Status := 0;
   STATUS[982].TimeStamp := 16#0000;
   STATUS[983].VALUE := 0.0;
   STATUS[983].TRIGVALUE := 0.0;
   STATUS[983].EXT.AlarmWarnUnAck := FALSE;
   STATUS[983].EXT.AckRequired := FALSE;
   STATUS[983].EXT.Maintanence := FALSE;
   STATUS[983].EXT.Operation := FALSE;
   STATUS[983].EXT.Forced := FALSE;
   STATUS[983].EXT.BIT29 := FALSE;
   STATUS[983].EXT.BIT30 := FALSE;
   STATUS[983].EXT.BIT31 := FALSE;
   STATUS[983].EXT.ModeBit1 := FALSE;
   STATUS[983].EXT.ModeBit2 := FALSE;
   STATUS[983].EXT.ModeBit3 := FALSE;
   STATUS[983].EXT.BIT19 := FALSE;
   STATUS[983].EXT.BIT20 := FALSE;
   STATUS[983].EXT.AlarmSuppressed := FALSE;
   STATUS[983].EXT.AlarmPrsent := FALSE;
   STATUS[983].EXT.AlarmFailUnAck := FALSE;
   STATUS[983].Status := 0;
   STATUS[983].TimeStamp := 16#0000;
   STATUS[984].VALUE := 0.0;
   STATUS[984].TRIGVALUE := 0.0;
   STATUS[984].EXT.AlarmWarnUnAck := FALSE;
   STATUS[984].EXT.AckRequired := FALSE;
   STATUS[984].EXT.Maintanence := FALSE;
   STATUS[984].EXT.Operation := FALSE;
   STATUS[984].EXT.Forced := FALSE;
   STATUS[984].EXT.BIT29 := FALSE;
   STATUS[984].EXT.BIT30 := FALSE;
   STATUS[984].EXT.BIT31 := FALSE;
   STATUS[984].EXT.ModeBit1 := FALSE;
   STATUS[984].EXT.ModeBit2 := FALSE;
   STATUS[984].EXT.ModeBit3 := FALSE;
   STATUS[984].EXT.BIT19 := FALSE;
   STATUS[984].EXT.BIT20 := FALSE;
   STATUS[984].EXT.AlarmSuppressed := FALSE;
   STATUS[984].EXT.AlarmPrsent := FALSE;
   STATUS[984].EXT.AlarmFailUnAck := FALSE;
   STATUS[984].Status := 0;
   STATUS[984].TimeStamp := 16#0000;
   STATUS[985].VALUE := 0.0;
   STATUS[985].TRIGVALUE := 0.0;
   STATUS[985].EXT.AlarmWarnUnAck := FALSE;
   STATUS[985].EXT.AckRequired := FALSE;
   STATUS[985].EXT.Maintanence := FALSE;
   STATUS[985].EXT.Operation := FALSE;
   STATUS[985].EXT.Forced := FALSE;
   STATUS[985].EXT.BIT29 := FALSE;
   STATUS[985].EXT.BIT30 := FALSE;
   STATUS[985].EXT.BIT31 := FALSE;
   STATUS[985].EXT.ModeBit1 := FALSE;
   STATUS[985].EXT.ModeBit2 := FALSE;
   STATUS[985].EXT.ModeBit3 := FALSE;
   STATUS[985].EXT.BIT19 := FALSE;
   STATUS[985].EXT.BIT20 := FALSE;
   STATUS[985].EXT.AlarmSuppressed := FALSE;
   STATUS[985].EXT.AlarmPrsent := FALSE;
   STATUS[985].EXT.AlarmFailUnAck := FALSE;
   STATUS[985].Status := 0;
   STATUS[985].TimeStamp := 16#0000;
   STATUS[986].VALUE := 0.0;
   STATUS[986].TRIGVALUE := 0.0;
   STATUS[986].EXT.AlarmWarnUnAck := FALSE;
   STATUS[986].EXT.AckRequired := FALSE;
   STATUS[986].EXT.Maintanence := FALSE;
   STATUS[986].EXT.Operation := FALSE;
   STATUS[986].EXT.Forced := FALSE;
   STATUS[986].EXT.BIT29 := FALSE;
   STATUS[986].EXT.BIT30 := FALSE;
   STATUS[986].EXT.BIT31 := FALSE;
   STATUS[986].EXT.ModeBit1 := FALSE;
   STATUS[986].EXT.ModeBit2 := FALSE;
   STATUS[986].EXT.ModeBit3 := FALSE;
   STATUS[986].EXT.BIT19 := FALSE;
   STATUS[986].EXT.BIT20 := FALSE;
   STATUS[986].EXT.AlarmSuppressed := FALSE;
   STATUS[986].EXT.AlarmPrsent := FALSE;
   STATUS[986].EXT.AlarmFailUnAck := FALSE;
   STATUS[986].Status := 0;
   STATUS[986].TimeStamp := 16#0000;
   STATUS[987].VALUE := 0.0;
   STATUS[987].TRIGVALUE := 0.0;
   STATUS[987].EXT.AlarmWarnUnAck := FALSE;
   STATUS[987].EXT.AckRequired := FALSE;
   STATUS[987].EXT.Maintanence := FALSE;
   STATUS[987].EXT.Operation := FALSE;
   STATUS[987].EXT.Forced := FALSE;
   STATUS[987].EXT.BIT29 := FALSE;
   STATUS[987].EXT.BIT30 := FALSE;
   STATUS[987].EXT.BIT31 := FALSE;
   STATUS[987].EXT.ModeBit1 := FALSE;
   STATUS[987].EXT.ModeBit2 := FALSE;
   STATUS[987].EXT.ModeBit3 := FALSE;
   STATUS[987].EXT.BIT19 := FALSE;
   STATUS[987].EXT.BIT20 := FALSE;
   STATUS[987].EXT.AlarmSuppressed := FALSE;
   STATUS[987].EXT.AlarmPrsent := FALSE;
   STATUS[987].EXT.AlarmFailUnAck := FALSE;
   STATUS[987].Status := 0;
   STATUS[987].TimeStamp := 16#0000;
   STATUS[988].VALUE := 0.0;
   STATUS[988].TRIGVALUE := 0.0;
   STATUS[988].EXT.AlarmWarnUnAck := FALSE;
   STATUS[988].EXT.AckRequired := FALSE;
   STATUS[988].EXT.Maintanence := FALSE;
   STATUS[988].EXT.Operation := FALSE;
   STATUS[988].EXT.Forced := FALSE;
   STATUS[988].EXT.BIT29 := FALSE;
   STATUS[988].EXT.BIT30 := FALSE;
   STATUS[988].EXT.BIT31 := FALSE;
   STATUS[988].EXT.ModeBit1 := FALSE;
   STATUS[988].EXT.ModeBit2 := FALSE;
   STATUS[988].EXT.ModeBit3 := FALSE;
   STATUS[988].EXT.BIT19 := FALSE;
   STATUS[988].EXT.BIT20 := FALSE;
   STATUS[988].EXT.AlarmSuppressed := FALSE;
   STATUS[988].EXT.AlarmPrsent := FALSE;
   STATUS[988].EXT.AlarmFailUnAck := FALSE;
   STATUS[988].Status := 0;
   STATUS[988].TimeStamp := 16#0000;
   STATUS[989].VALUE := 0.0;
   STATUS[989].TRIGVALUE := 0.0;
   STATUS[989].EXT.AlarmWarnUnAck := FALSE;
   STATUS[989].EXT.AckRequired := FALSE;
   STATUS[989].EXT.Maintanence := FALSE;
   STATUS[989].EXT.Operation := FALSE;
   STATUS[989].EXT.Forced := FALSE;
   STATUS[989].EXT.BIT29 := FALSE;
   STATUS[989].EXT.BIT30 := FALSE;
   STATUS[989].EXT.BIT31 := FALSE;
   STATUS[989].EXT.ModeBit1 := FALSE;
   STATUS[989].EXT.ModeBit2 := FALSE;
   STATUS[989].EXT.ModeBit3 := FALSE;
   STATUS[989].EXT.BIT19 := FALSE;
   STATUS[989].EXT.BIT20 := FALSE;
   STATUS[989].EXT.AlarmSuppressed := FALSE;
   STATUS[989].EXT.AlarmPrsent := FALSE;
   STATUS[989].EXT.AlarmFailUnAck := FALSE;
   STATUS[989].Status := 0;
   STATUS[989].TimeStamp := 16#0000;
   STATUS[990].VALUE := 0.0;
   STATUS[990].TRIGVALUE := 0.0;
   STATUS[990].EXT.AlarmWarnUnAck := FALSE;
   STATUS[990].EXT.AckRequired := FALSE;
   STATUS[990].EXT.Maintanence := FALSE;
   STATUS[990].EXT.Operation := FALSE;
   STATUS[990].EXT.Forced := FALSE;
   STATUS[990].EXT.BIT29 := FALSE;
   STATUS[990].EXT.BIT30 := FALSE;
   STATUS[990].EXT.BIT31 := FALSE;
   STATUS[990].EXT.ModeBit1 := FALSE;
   STATUS[990].EXT.ModeBit2 := FALSE;
   STATUS[990].EXT.ModeBit3 := FALSE;
   STATUS[990].EXT.BIT19 := FALSE;
   STATUS[990].EXT.BIT20 := FALSE;
   STATUS[990].EXT.AlarmSuppressed := FALSE;
   STATUS[990].EXT.AlarmPrsent := FALSE;
   STATUS[990].EXT.AlarmFailUnAck := FALSE;
   STATUS[990].Status := 0;
   STATUS[990].TimeStamp := 16#0000;
   STATUS[991].VALUE := 0.0;
   STATUS[991].TRIGVALUE := 0.0;
   STATUS[991].EXT.AlarmWarnUnAck := FALSE;
   STATUS[991].EXT.AckRequired := FALSE;
   STATUS[991].EXT.Maintanence := FALSE;
   STATUS[991].EXT.Operation := FALSE;
   STATUS[991].EXT.Forced := FALSE;
   STATUS[991].EXT.BIT29 := FALSE;
   STATUS[991].EXT.BIT30 := FALSE;
   STATUS[991].EXT.BIT31 := FALSE;
   STATUS[991].EXT.ModeBit1 := FALSE;
   STATUS[991].EXT.ModeBit2 := FALSE;
   STATUS[991].EXT.ModeBit3 := FALSE;
   STATUS[991].EXT.BIT19 := FALSE;
   STATUS[991].EXT.BIT20 := FALSE;
   STATUS[991].EXT.AlarmSuppressed := FALSE;
   STATUS[991].EXT.AlarmPrsent := FALSE;
   STATUS[991].EXT.AlarmFailUnAck := FALSE;
   STATUS[991].Status := 0;
   STATUS[991].TimeStamp := 16#0000;
   STATUS[992].VALUE := 0.0;
   STATUS[992].TRIGVALUE := 0.0;
   STATUS[992].EXT.AlarmWarnUnAck := FALSE;
   STATUS[992].EXT.AckRequired := FALSE;
   STATUS[992].EXT.Maintanence := FALSE;
   STATUS[992].EXT.Operation := FALSE;
   STATUS[992].EXT.Forced := FALSE;
   STATUS[992].EXT.BIT29 := FALSE;
   STATUS[992].EXT.BIT30 := FALSE;
   STATUS[992].EXT.BIT31 := FALSE;
   STATUS[992].EXT.ModeBit1 := FALSE;
   STATUS[992].EXT.ModeBit2 := FALSE;
   STATUS[992].EXT.ModeBit3 := FALSE;
   STATUS[992].EXT.BIT19 := FALSE;
   STATUS[992].EXT.BIT20 := FALSE;
   STATUS[992].EXT.AlarmSuppressed := FALSE;
   STATUS[992].EXT.AlarmPrsent := FALSE;
   STATUS[992].EXT.AlarmFailUnAck := FALSE;
   STATUS[992].Status := 0;
   STATUS[992].TimeStamp := 16#0000;
   STATUS[993].VALUE := 0.0;
   STATUS[993].TRIGVALUE := 0.0;
   STATUS[993].EXT.AlarmWarnUnAck := FALSE;
   STATUS[993].EXT.AckRequired := FALSE;
   STATUS[993].EXT.Maintanence := FALSE;
   STATUS[993].EXT.Operation := FALSE;
   STATUS[993].EXT.Forced := FALSE;
   STATUS[993].EXT.BIT29 := FALSE;
   STATUS[993].EXT.BIT30 := FALSE;
   STATUS[993].EXT.BIT31 := FALSE;
   STATUS[993].EXT.ModeBit1 := FALSE;
   STATUS[993].EXT.ModeBit2 := FALSE;
   STATUS[993].EXT.ModeBit3 := FALSE;
   STATUS[993].EXT.BIT19 := FALSE;
   STATUS[993].EXT.BIT20 := FALSE;
   STATUS[993].EXT.AlarmSuppressed := FALSE;
   STATUS[993].EXT.AlarmPrsent := FALSE;
   STATUS[993].EXT.AlarmFailUnAck := FALSE;
   STATUS[993].Status := 0;
   STATUS[993].TimeStamp := 16#0000;
   STATUS[994].VALUE := 0.0;
   STATUS[994].TRIGVALUE := 0.0;
   STATUS[994].EXT.AlarmWarnUnAck := FALSE;
   STATUS[994].EXT.AckRequired := FALSE;
   STATUS[994].EXT.Maintanence := FALSE;
   STATUS[994].EXT.Operation := FALSE;
   STATUS[994].EXT.Forced := FALSE;
   STATUS[994].EXT.BIT29 := FALSE;
   STATUS[994].EXT.BIT30 := FALSE;
   STATUS[994].EXT.BIT31 := FALSE;
   STATUS[994].EXT.ModeBit1 := FALSE;
   STATUS[994].EXT.ModeBit2 := FALSE;
   STATUS[994].EXT.ModeBit3 := FALSE;
   STATUS[994].EXT.BIT19 := FALSE;
   STATUS[994].EXT.BIT20 := FALSE;
   STATUS[994].EXT.AlarmSuppressed := FALSE;
   STATUS[994].EXT.AlarmPrsent := FALSE;
   STATUS[994].EXT.AlarmFailUnAck := FALSE;
   STATUS[994].Status := 0;
   STATUS[994].TimeStamp := 16#0000;
   STATUS[995].VALUE := 0.0;
   STATUS[995].TRIGVALUE := 0.0;
   STATUS[995].EXT.AlarmWarnUnAck := FALSE;
   STATUS[995].EXT.AckRequired := FALSE;
   STATUS[995].EXT.Maintanence := FALSE;
   STATUS[995].EXT.Operation := FALSE;
   STATUS[995].EXT.Forced := FALSE;
   STATUS[995].EXT.BIT29 := FALSE;
   STATUS[995].EXT.BIT30 := FALSE;
   STATUS[995].EXT.BIT31 := FALSE;
   STATUS[995].EXT.ModeBit1 := FALSE;
   STATUS[995].EXT.ModeBit2 := FALSE;
   STATUS[995].EXT.ModeBit3 := FALSE;
   STATUS[995].EXT.BIT19 := FALSE;
   STATUS[995].EXT.BIT20 := FALSE;
   STATUS[995].EXT.AlarmSuppressed := FALSE;
   STATUS[995].EXT.AlarmPrsent := FALSE;
   STATUS[995].EXT.AlarmFailUnAck := FALSE;
   STATUS[995].Status := 0;
   STATUS[995].TimeStamp := 16#0000;
   STATUS[996].VALUE := 0.0;
   STATUS[996].TRIGVALUE := 0.0;
   STATUS[996].EXT.AlarmWarnUnAck := FALSE;
   STATUS[996].EXT.AckRequired := FALSE;
   STATUS[996].EXT.Maintanence := FALSE;
   STATUS[996].EXT.Operation := FALSE;
   STATUS[996].EXT.Forced := FALSE;
   STATUS[996].EXT.BIT29 := FALSE;
   STATUS[996].EXT.BIT30 := FALSE;
   STATUS[996].EXT.BIT31 := FALSE;
   STATUS[996].EXT.ModeBit1 := FALSE;
   STATUS[996].EXT.ModeBit2 := FALSE;
   STATUS[996].EXT.ModeBit3 := FALSE;
   STATUS[996].EXT.BIT19 := FALSE;
   STATUS[996].EXT.BIT20 := FALSE;
   STATUS[996].EXT.AlarmSuppressed := FALSE;
   STATUS[996].EXT.AlarmPrsent := FALSE;
   STATUS[996].EXT.AlarmFailUnAck := FALSE;
   STATUS[996].Status := 0;
   STATUS[996].TimeStamp := 16#0000;
   STATUS[997].VALUE := 0.0;
   STATUS[997].TRIGVALUE := 0.0;
   STATUS[997].EXT.AlarmWarnUnAck := FALSE;
   STATUS[997].EXT.AckRequired := FALSE;
   STATUS[997].EXT.Maintanence := FALSE;
   STATUS[997].EXT.Operation := FALSE;
   STATUS[997].EXT.Forced := FALSE;
   STATUS[997].EXT.BIT29 := FALSE;
   STATUS[997].EXT.BIT30 := FALSE;
   STATUS[997].EXT.BIT31 := FALSE;
   STATUS[997].EXT.ModeBit1 := FALSE;
   STATUS[997].EXT.ModeBit2 := FALSE;
   STATUS[997].EXT.ModeBit3 := FALSE;
   STATUS[997].EXT.BIT19 := FALSE;
   STATUS[997].EXT.BIT20 := FALSE;
   STATUS[997].EXT.AlarmSuppressed := FALSE;
   STATUS[997].EXT.AlarmPrsent := FALSE;
   STATUS[997].EXT.AlarmFailUnAck := FALSE;
   STATUS[997].Status := 0;
   STATUS[997].TimeStamp := 16#0000;
   STATUS[998].VALUE := 0.0;
   STATUS[998].TRIGVALUE := 0.0;
   STATUS[998].EXT.AlarmWarnUnAck := FALSE;
   STATUS[998].EXT.AckRequired := FALSE;
   STATUS[998].EXT.Maintanence := FALSE;
   STATUS[998].EXT.Operation := FALSE;
   STATUS[998].EXT.Forced := FALSE;
   STATUS[998].EXT.BIT29 := FALSE;
   STATUS[998].EXT.BIT30 := FALSE;
   STATUS[998].EXT.BIT31 := FALSE;
   STATUS[998].EXT.ModeBit1 := FALSE;
   STATUS[998].EXT.ModeBit2 := FALSE;
   STATUS[998].EXT.ModeBit3 := FALSE;
   STATUS[998].EXT.BIT19 := FALSE;
   STATUS[998].EXT.BIT20 := FALSE;
   STATUS[998].EXT.AlarmSuppressed := FALSE;
   STATUS[998].EXT.AlarmPrsent := FALSE;
   STATUS[998].EXT.AlarmFailUnAck := FALSE;
   STATUS[998].Status := 0;
   STATUS[998].TimeStamp := 16#0000;
   STATUS[999].VALUE := 0.0;
   STATUS[999].TRIGVALUE := 0.0;
   STATUS[999].EXT.AlarmWarnUnAck := FALSE;
   STATUS[999].EXT.AckRequired := FALSE;
   STATUS[999].EXT.Maintanence := FALSE;
   STATUS[999].EXT.Operation := FALSE;
   STATUS[999].EXT.Forced := FALSE;
   STATUS[999].EXT.BIT29 := FALSE;
   STATUS[999].EXT.BIT30 := FALSE;
   STATUS[999].EXT.BIT31 := FALSE;
   STATUS[999].EXT.ModeBit1 := FALSE;
   STATUS[999].EXT.ModeBit2 := FALSE;
   STATUS[999].EXT.ModeBit3 := FALSE;
   STATUS[999].EXT.BIT19 := FALSE;
   STATUS[999].EXT.BIT20 := FALSE;
   STATUS[999].EXT.AlarmSuppressed := FALSE;
   STATUS[999].EXT.AlarmPrsent := FALSE;
   STATUS[999].EXT.AlarmFailUnAck := FALSE;
   STATUS[999].Status := 0;
   STATUS[999].TimeStamp := 16#0000;
   STATUS[1000].VALUE := 0.0;
   STATUS[1000].TRIGVALUE := 0.0;
   STATUS[1000].EXT.AlarmWarnUnAck := FALSE;
   STATUS[1000].EXT.AckRequired := FALSE;
   STATUS[1000].EXT.Maintanence := FALSE;
   STATUS[1000].EXT.Operation := FALSE;
   STATUS[1000].EXT.Forced := FALSE;
   STATUS[1000].EXT.BIT29 := FALSE;
   STATUS[1000].EXT.BIT30 := FALSE;
   STATUS[1000].EXT.BIT31 := FALSE;
   STATUS[1000].EXT.ModeBit1 := FALSE;
   STATUS[1000].EXT.ModeBit2 := FALSE;
   STATUS[1000].EXT.ModeBit3 := FALSE;
   STATUS[1000].EXT.BIT19 := FALSE;
   STATUS[1000].EXT.BIT20 := FALSE;
   STATUS[1000].EXT.AlarmSuppressed := FALSE;
   STATUS[1000].EXT.AlarmPrsent := FALSE;
   STATUS[1000].EXT.AlarmFailUnAck := FALSE;
   STATUS[1000].Status := 0;
   STATUS[1000].TimeStamp := 16#0000;
END_DATA_BLOCK

